(* System generated code, could be modified for your application *)
	c_udiNumberOfSubModules			: UDINT := 4;			(* Number of SubModules: Added extra 1 for Crank Module *)
	c_udiSlave3						: UDINT := 1;
	c_udiSlave4						: UDINT := 2;
	c_udiCrank						: UDINT := 4;			(* special constant for Crank module *)
	c_udiNocke1						: UDINT := 3;
(* End of system generated code, could be modified for your application *)
END_VAR

VAR (* User specific variables *)
	stSlave3Interface				: AXM.ST_ModuleInterface;
	fbSlave3Module					: AXM.FB_AxisModule;
	
	stSlave4Interface				: AXM.ST_ModuleInterface;
	fbSlave4Module					: AXM.FB_AxisModule;

	fbAxisModuleController			: AXM.FB_AxisModuleController;

	stNocke1Interface				: ST_ExampleLeafModuleInterface;
	fbNocke1Module					: FB_ExampleLeafModule;

	fbExampleLeafModuleController	: FB_ExampleLeafModuleController;
	
	(*included for CrankModule*)
	stCrankModuleItf			: CRKM.ST_ModuleInterface;
	fbCrankModule				: CRKM.FB_CrankModule;
	fbCrankModuleCtrl			: CRKM.FB_CrankModuleController;
	
	(*included for CrankModule*)
	
	xFirstCall						: BOOL := TRUE;
	iPosState						: INT := 1;
END_VAR

VAR_INPUT
(* Master of AlphaModule *)
	i_ifMaster						: SystemConfigurationItf.IF_Master;
END_VAR

VAR_IN_OUT
(* TPL.ST_StandardModuleInterface *)
	iq_stStandardModuleItf			: TPL.ST_StandardModuleInterface;
	
(* TPL.ST_StandardMotionInterface *)
	iq_stStandardMotionItf			: TPL.ST_StandardMotionInterface;
	
(* ExceptionHandling and Logging *)	
	iq_stExceptionList				: TPL.ST_ExceptionList;
	iq_stLogDataList				: TPL.ST_LogDataList;
END_VAR

VAR
	xInitSuccessful : BOOL := TRUE;
	
(* Standard related variables *)
	astSubModuleInterface			: ARRAY[1..c_udiNumberOfSubModules] OF TPL.ST_StandardModuleInterface;		(* Interface to modules *)
	aaudiSubModuleGroups			: ARRAY[1..c_udiNumberOfGroups,1..c_udiNumberOfGroupMembers] OF UDINT;
	adwSubModuleAddInterfaces		: ARRAY[1..c_udiNumberOfSubModules] OF DWORD;

(* Modules related variables *)
	fbModuleController				: TPL.FB_ModuleController;
	etDiagModuleController			: GD.ET_Diag;
	etDiagExtModuleController		: TPL.ET_DiagExt;
	sMsgModuleController			: STRING[80];
	xWaitForStartStep				: BOOL;

	astListOfCmdTables				: ARRAY [1..c_udiNumberOfCmdTables] OF TPL.ST_CmdTable;
	udiTableIndex					: UDINT;
	udiStepIndex					: UDINT;
	diStep							: DINT;

	astPrepareTable					: ARRAY [1..c_udiNumberOfCmdSteps] OF TPL.ST_Cmd;		(* Relating  Cmd table *)
	astAutoTable					: ARRAY [1..c_udiNumberOfCmdSteps] OF TPL.ST_Cmd;		(* Relating  Cmd table *)
	astManualTable					: ARRAY [1..c_udiNumberOfCmdSteps] OF TPL.ST_Cmd;		(* Relating  Cmd table *)
	astHoldTable					: ARRAY [1..c_udiNumberOfCmdSteps] OF TPL.ST_Cmd;		(* Relating  Cmd table *)
	astStartTable					: ARRAY [1..c_udiNumberOfCmdSteps] OF TPL.ST_Cmd;		(* Relating  Cmd table *)
	astStopTable					: ARRAY [1..c_udiNumberOfCmdSteps] OF TPL.ST_Cmd;		(* Relating  Cmd table *)
	astBrakeReleaseTable			: ARRAY [1..c_udiNumberOfCmdSteps] OF TPL.ST_Cmd;		(* Relating  Cmd table *)
	astAbortTable					: ARRAY [1..c_udiNumberOfCmdSteps] OF TPL.ST_Cmd;		(* Relating  Cmd table *)

(* ExceptionHandling related variables *)
	fbExceptionHandler				: TPL.FB_ExceptionHandler;

	aetReactionTranslationMode		: ARRAY[1..c_udiNumberOfSubModules] OF TPL.ET_ReactionTranslationMode;
	aastReactionTranslationTable	: ARRAY[1..c_udiNumberOfSubModules,1..TPL.Gc_udiMaxNumberOfReactions] OF TPL.ST_Reaction;
	astReactionTranslationJobs		: ARRAY[1..c_udiNumberOfSubModules] OF TPL.ST_ReactionTranslationJobs;
	
(* Exception declaration *)
	stUserException1				: TPL.ST_Exception;
	stUserException2				: TPL.ST_Exception;
	xModuleUserException1			: BOOL;
	xModuleUserException2			: BOOL;
	
	stUpdateStructsException		: TPL.ST_Exception;
	xUpdateStructsException			: BOOL;
	
	stInitReactionsException		: TPL.ST_Exception;
	xInitReactionsException			: BOOL;
	
	stInitSubModulesException		: TPL.ST_Exception;
	xInitSubModulesException		: BOOL;
	
	stIsDriveVirtualException		: TPL.ST_Exception;
	xIsDriveVirtualException		: BOOL;
	
(* Logging related variables*)
	fbLogger						: TPL.FB_Logger;

(* OnlineChange related variables *)
	fbDetectOnlineChange			: TPL.FB_DetectOnlineChange;
	xDetectOnlineChangeActive		: BOOL; 
	xDetectOnlineChangeReady		: BOOL; 
	etDetectOnlineChangeDiag		: GD.ET_Diag;
	etDetectOnlineChangeDiagExt		: TPL.ET_DiagExt; 
	sDetectOnlineChangeMsg			: STRING[80];
	
(* Init related variables *)		
	stLogicalAddressMaster			: SystemConfigurationItf.ST_LogicalAddress;
	lrShaftRefDelay					: LREAL;
	diResult						: DINT;	
	
	xDriveIsVirtual					: BOOL;	

(* POU-Feedback related variables*)	
	etDiag			: GD.ET_Diag;
	etDiagExt		: ET_DiagExt;
	etDiagDiagExtExampleLeafModule		: ET_DiagExtExampleLeafModule;
	etDiagExtTPL	: TPL.ET_DiagExt;
	etDiagExtAXM	: AXM.ET_DiagExt;
	etDiagExtCRKM	: CRKM.ET_DiagExt;
	sMsgBuffer		: STRING[80];
END_VAR

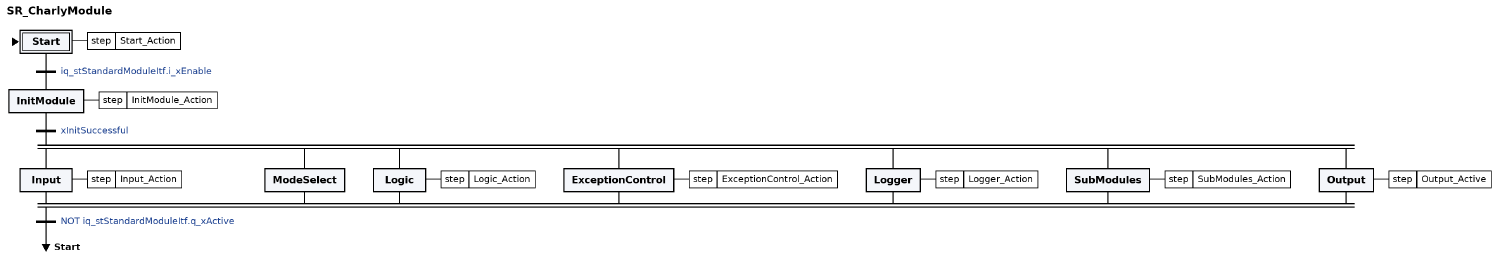
INITIAL_STEP Start:
    Start_Action(N);  // step action
END_STEP
TRANSITION FROM Start TO InitModule
    := iq_stStandardModuleItf.i_xEnable;
END_TRANSITION
STEP InitModule:
    InitModule_Action(N);  // step action
END_STEP
TRANSITION FROM InitModule TO (Input, ModeSelect, Logic, ExceptionControl, Logger, SubModules, Output)
    := xInitSuccessful;
END_TRANSITION
STEP Input:
    Input_Action(N);  // step action
END_STEP
STEP ModeSelect:
END_STEP
STEP Logic:
    Logic_Action(N);  // step action
END_STEP
STEP ExceptionControl:
    ExceptionControl_Action(N);  // step action
END_STEP
STEP Logger:
    Logger_Action(N);  // step action
END_STEP
STEP SubModules:
    SubModules_Action(N);  // step action
END_STEP
STEP Output:
    Output_Active(N);  // step action
END_STEP
TRANSITION FROM (Input, ModeSelect, Logic, ExceptionControl, Logger, SubModules, Output) TO Start
    := NOT iq_stStandardModuleItf.q_xActive;
END_TRANSITION

ACTION ExceptionControl_Action:
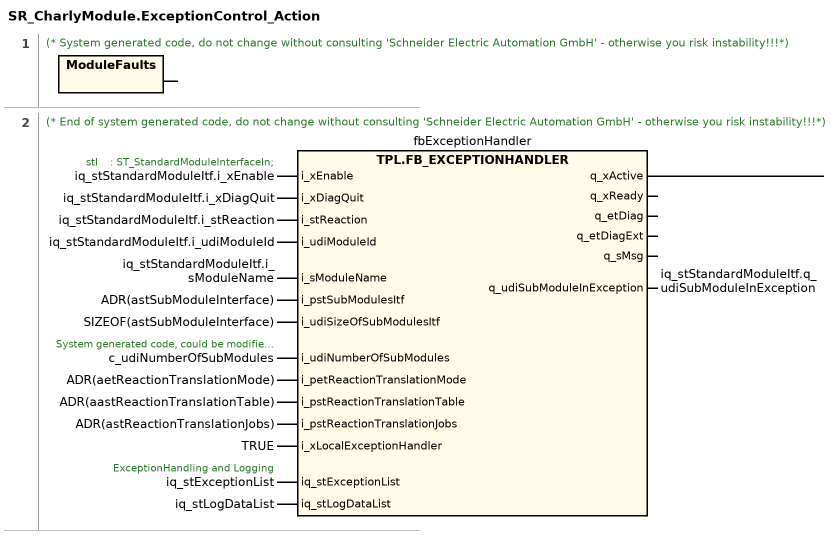
// NETWORK 1
// (* System generated code, do not change without consulting 'Schneider Electric Automation GmbH' - otherwise you risk instability!!!*)
ModuleFaults();

// NETWORK 2
// (* End of system generated code, do not change without consulting 'Schneider Electric Automation GmbH' - otherwise you risk instability!!!*)
//   fbExceptionHandler: ExceptionHandling related variables
//   iq_stStandardModuleItf.i_xEnable: stI : ST_StandardModuleInterfaceIn;
//   c_udiNumberOfSubModules: System generated code, could be modified for your application
//   iq_stExceptionList: ExceptionHandling and Logging
fbExceptionHandler(
    i_xEnable := iq_stStandardModuleItf.i_xEnable,
    i_xDiagQuit := iq_stStandardModuleItf.i_xDiagQuit,
    i_stReaction := iq_stStandardModuleItf.i_stReaction,
    i_udiModuleId := iq_stStandardModuleItf.i_udiModuleId,
    i_sModuleName := iq_stStandardModuleItf.i_sModuleName,
    i_pstSubModulesItf := ADR(astSubModuleInterface),
    i_udiSizeOfSubModulesItf := SIZEOF(astSubModuleInterface),
    i_udiNumberOfSubModules := c_udiNumberOfSubModules,
    i_petReactionTranslationMode := ADR(aetReactionTranslationMode),
    i_pstReactionTranslationTable := ADR(aastReactionTranslationTable),
    i_pstReactionTranslationJobs := ADR(astReactionTranslationJobs),
    i_xLocalExceptionHandler := TRUE,
    iq_stExceptionList := iq_stExceptionList,
    iq_stLogDataList := iq_stLogDataList,
    q_udiSubModuleInException => iq_stStandardModuleItf.q_udiSubModuleInException); // TPL.FB_EXCEPTIONHANDLER
END_ACTION

ACTION Init_CmdTables:
(* System generated code, could be modified for your application *)

(*********************************************************************************************************************)
(*** Prepare/Homing  ***)

TPL.FC_FirstStep(udiStepIndex, diStep);
astPrepareTable[udiStepIndex].sTitle					:= 'DriveEnable CrankModule';
astPrepareTable[udiStepIndex].udiModuleName				:= c_udiCrank;
astPrepareTable[udiStepIndex].diStep					:= diStep;
astPrepareTable[udiStepIndex].diCMD						:= CRKM.ET_Cmd.DriveEnableOn;
astPrepareTable[udiStepIndex].timTimeOut				:= T#0MS;
astPrepareTable[udiStepIndex].xEndCMD					:= FALSE;

TPL.FC_NextStep(udiStepIndex, diStep);
astPrepareTable[udiStepIndex].sTitle					:= 'Homing Mode CrankModule';
astPrepareTable[udiStepIndex].udiModuleName				:= c_udiCrank;
astPrepareTable[udiStepIndex].diStep					:= diStep;
astPrepareTable[udiStepIndex].diCMD						:= CRKM.ET_Cmd.Homing;
astPrepareTable[udiStepIndex].timTimeOut				:= T#0MS;
astPrepareTable[udiStepIndex].xEndCMD					:= FALSE;

TPL.FC_NextStep(udiStepIndex, diStep);
astPrepareTable[udiStepIndex].sTitle					:= 'Start CrankModule';
astPrepareTable[udiStepIndex].udiModuleName				:= c_udiCrank;
astPrepareTable[udiStepIndex].diStep					:= diStep;
astPrepareTable[udiStepIndex].diCMD						:= CRKM.ET_Cmd.Start;
astPrepareTable[udiStepIndex].timTimeOut				:= T#0MS;
astPrepareTable[udiStepIndex].xEndCMD					:= FALSE;

TPL.FC_LastStep(udiStepIndex, diStep);
astPrepareTable[udiStepIndex].sTitle					:= 'End';
astPrepareTable[udiStepIndex].udiModuleName				:= 0;
astPrepareTable[udiStepIndex].diStep					:= diStep;
astPrepareTable[udiStepIndex].diCMD						:= 0;
astPrepareTable[udiStepIndex].timTimeOut				:= T#0MS;
astPrepareTable[udiStepIndex].xEndCMD					:= TRUE;

TPL.FC_FirstCmdTable(iq_udiTableIndex:= udiTableIndex);
astListofCMDTables[udiTableIndex].sTitle				:= 'Prepare';
astListofCMDTables[udiTableIndex].diCMD					:= ET_Cmd.Prepare;
astListofCMDTables[udiTableIndex].udiNumberOfCmdSteps	:= udiStepIndex;

(*********************************************************************************************************************)
(*** Auto/Endless  ***)


TPL.FC_FirstStep(udiStepIndex, diStep);
astAutoTable[udiStepIndex].sTitle						:= 'DriveEnable CrankModule';
astAutoTable[udiStepIndex].udiModuleName				:= c_udiCrank;
astAutoTable[udiStepIndex].diStep						:= diStep;
astAutoTable[udiStepIndex].diCMD						:= CRKM.ET_Cmd.DriveEnableOn;
astAutoTable[udiStepIndex].timTimeOut					:= T#0MS;
astAutoTable[udiStepIndex].xEndCMD						:= FALSE;

TPL.FC_NextStep(udiStepIndex, diStep);
astAutoTable[udiStepIndex].sTitle						:= 'Auto/Endless CrankModule';
astAutoTable[udiStepIndex].udiModuleName				:= c_udiCrank;
astAutoTable[udiStepIndex].diStep						:= diStep;
astAutoTable[udiStepIndex].diCMD						:= CRKM.ET_Cmd.Endless;
astAutoTable[udiStepIndex].timTimeOut					:= T#0MS;
astAutoTable[udiStepIndex].xEndCMD						:= FALSE;

TPL.FC_NextStep(udiStepIndex, diStep);
astAutoTable[udiStepIndex].sTitle						:= 'Start CrankModule';
astAutoTable[udiStepIndex].udiModuleName				:= c_udiCrank;
astAutoTable[udiStepIndex].diStep						:= diStep;
astAutoTable[udiStepIndex].diCMD						:= CRKM.ET_Cmd.Start;
astAutoTable[udiStepIndex].timTimeOut					:= T#0MS;
astAutoTable[udiStepIndex].xEndCMD						:= FALSE;

TPL.FC_NextStep(udiStepIndex, diStep);
astAutoTable[udiStepIndex].sTitle						:= 'Endless Mode Slave3';
astAutoTable[udiStepIndex].udiModuleName				:= c_udiSlave3;
astAutoTable[udiStepIndex].diStep						:= diStep;
astAutoTable[udiStepIndex].diCMD						:= AXM.ET_Cmd.Endless; 
astAutoTable[udiStepIndex].timTimeOut					:= T#0MS;
astAutoTable[udiStepIndex].xEndCMD						:= FALSE;

TPL.FC_NextStep(udiStepIndex, diStep);
astAutoTable[udiStepIndex].sTitle						:= 'Positioning Mode Slave4';
astAutoTable[udiStepIndex].udiModuleName				:= c_udiSlave4;
astAutoTable[udiStepIndex].diStep						:= diStep;
astAutoTable[udiStepIndex].diCMD						:= AXM.ET_Cmd.Positioning;
astAutoTable[udiStepIndex].timTimeOut					:= T#0MS;
astAutoTable[udiStepIndex].xEndCMD						:= FALSE;

TPL.FC_NextStep(udiStepIndex, diStep);
astAutoTable[udiStepIndex].sTitle						:= 'Start Slave3';
astAutoTable[udiStepIndex].udiModuleName				:= c_udiSlave3;
astAutoTable[udiStepIndex].diStep						:= diStep;
astAutoTable[udiStepIndex].diCMD						:= AXM.ET_Cmd.Start;
astAutoTable[udiStepIndex].timTimeOut					:= T#0MS;
astAutoTable[udiStepIndex].xEndCMD						:= FALSE;



TPL.FC_LastStep(udiStepIndex, diStep);
astAutoTable[udiStepIndex].sTitle						:= 'End';
astAutoTable[udiStepIndex].udiModuleName				:= 0;
astAutoTable[udiStepIndex].diStep						:= diStep;
astAutoTable[udiStepIndex].diCMD						:= 0;
astAutoTable[udiStepIndex].timTimeOut					:= T#0MS;
astAutoTable[udiStepIndex].xEndCMD						:= TRUE;

TPL.FC_NextCmdTable(iq_udiTableIndex:= udiTableIndex);
astListofCMDTables[udiTableIndex].sTitle				:= 'Auto';
astListofCMDTables[udiTableIndex].diCMD					:= ET_Cmd.Auto;
astListofCMDTables[udiTableIndex].udiNumberOfCmdSteps	:= udiStepIndex;


(*********************************************************************************************************************)
(*** Manual  ***)

TPL.FC_FirstStep(udiStepIndex, diStep);
astManualTable[udiStepIndex].sTitle						:= 'DriveEnable On CrankModule';
astManualTable[udiStepIndex].udiModuleName				:= c_udiCrank;
astManualTable[udiStepIndex].diStep						:= diStep;
astManualTable[udiStepIndex].diCMD						:= CRKM.ET_Cmd.DriveEnableOn;
astManualTable[udiStepIndex].timTimeOut					:= T#0MS;
astManualTable[udiStepIndex].xEndCMD					:= FALSE;

TPL.FC_NextStep(udiStepIndex, diStep);
astManualTable[udiStepIndex].sTitle						:= 'Manual Mode CrankModule';
astManualTable[udiStepIndex].udiModuleName				:= c_udiCrank;
astManualTable[udiStepIndex].diStep						:= diStep;
astManualTable[udiStepIndex].diCMD						:= CRKM.ET_Cmd.Manual;
astManualTable[udiStepIndex].timTimeOut					:= T#0MS;
astManualTable[udiStepIndex].xEndCMD					:= FALSE;

TPL.FC_LastStep(udiStepIndex, diStep);
astManualTable[udiStepIndex].sTitle						:= 'End';
astManualTable[udiStepIndex].udiModuleName				:= 0;
astManualTable[udiStepIndex].diStep						:= diStep;
astManualTable[udiStepIndex].diCMD						:= 0;
astManualTable[udiStepIndex].timTimeOut					:= T#0MS;
astManualTable[udiStepIndex].xEndCMD					:= TRUE;

TPL.FC_NextCmdTable(iq_udiTableIndex:= udiTableIndex);
astListofCMDTables[udiTableIndex].sTitle				:= 'Manual';
astListofCMDTables[udiTableIndex].diCMD					:= ET_Cmd.Manual;
astListofCMDTables[udiTableIndex].udiNumberOfCmdSteps	:= udiStepIndex;

(*********************************************************************************************************************)
(*** Stop ***)

TPL.FC_FirstStep(udiStepIndex, diStep);
astStopTable[udiStepIndex].sTitle						:= 'Stop CrankModule';
astStopTable[udiStepIndex].udiModuleName				:= c_udiCrank;
astStopTable[udiStepIndex].diStep						:= diStep;
astStopTable[udiStepIndex].diCMD						:= CRKM.ET_Cmd.Stop;
astStopTable[udiStepIndex].timTimeOut					:= T#0MS;
astStopTable[udiStepIndex].xEndCMD						:= FALSE;

TPL.FC_LastStep(udiStepIndex, diStep);
astStopTable[udiStepIndex].sTitle						:= 'End';
astStopTable[udiStepIndex].udiModuleName				:= 0;
astStopTable[udiStepIndex].diStep						:= diStep;
astStopTable[udiStepIndex].diCMD						:= 0;
astStopTable[udiStepIndex].timTimeOut					:= T#0MS;
astStopTable[udiStepIndex].xEndCMD						:= TRUE;

TPL.FC_NextCmdTable(iq_udiTableIndex:= udiTableIndex);
astListofCMDTables[udiTableIndex].sTitle				:= 'Stop';
astListofCMDTables[udiTableIndex].diCMD					:= ET_Cmd.Stop;
astListofCMDTables[udiTableIndex].udiNumberOfCmdSteps	:= udiStepIndex;

(*********************************************************************************************************************)
(*** Start ***)

TPL.FC_FirstStep(udiStepIndex, diStep);
astStartTable[udiStepIndex].sTitle						:= 'Start CrankModule';
astStartTable[udiStepIndex].udiModuleName				:= c_udiCrank;
astStartTable[udiStepIndex].diStep						:= diStep;
astStartTable[udiStepIndex].diCMD						:= CRKM.ET_Cmd.Start;
astStartTable[udiStepIndex].timTimeOut					:= T#0MS;
astStartTable[udiStepIndex].xEndCMD						:= FALSE;

TPL.FC_LastStep(udiStepIndex, diStep);
astStartTable[udiStepIndex].sTitle						:= 'End';
astStartTable[udiStepIndex].udiModuleName				:= 0;
astStartTable[udiStepIndex].diStep						:= diStep;
astStartTable[udiStepIndex].diCMD						:= 0;
astStartTable[udiStepIndex].timTimeOut					:= T#0MS;
astStartTable[udiStepIndex].xEndCMD						:= TRUE;

TPL.FC_NextCmdTable(iq_udiTableIndex:= udiTableIndex);
astListofCMDTables[udiTableIndex].sTitle				:= 'Start';
astListofCMDTables[udiTableIndex].diCMD					:= ET_Cmd.Start;
astListofCMDTables[udiTableIndex].udiNumberOfCmdSteps	:= udiStepIndex;

(*********************************************************************************************************************)
(*** Abort ***)

TPL.FC_FirstStep(udiStepIndex, diStep);
astAbortTable[udiStepIndex].sTitle						:= 'Stop CrankModule';
astAbortTable[udiStepIndex].udiModuleName				:= c_udiCrank;
astAbortTable[udiStepIndex].diStep						:= diStep;
astAbortTable[udiStepIndex].diCMD						:= CRKM.ET_Cmd.Stop;
astAbortTable[udiStepIndex].timTimeOut					:= T#0MS;
astAbortTable[udiStepIndex].xEndCMD						:= FALSE;

TPL.FC_LastStep(udiStepIndex, diStep);
astAbortTable[udiStepIndex].sTitle						:= 'End';
astAbortTable[udiStepIndex].udiModuleName				:= 0;
astAbortTable[udiStepIndex].diStep						:= diStep;
astAbortTable[udiStepIndex].diCMD						:= 0;
astAbortTable[udiStepIndex].timTimeOut					:= T#0MS;
astAbortTable[udiStepIndex].xEndCMD						:= TRUE;

TPL.FC_NextCmdTable(iq_udiTableIndex:= udiTableIndex);
astListofCMDTables[udiTableIndex].sTitle				:= 'Abort';
astListofCMDTables[udiTableIndex].diCMD					:= ET_Cmd.Abort;
astListofCMDTables[udiTableIndex].udiNumberOfCmdSteps	:= udiStepIndex;

(*********************************************************************************************************************)
(*** Hold ***)

TPL.FC_FirstStep(udiStepIndex, diStep);
astHoldTable[udiStepIndex].sTitle						:= 'Hold CrankModule';
astHoldTable[udiStepIndex].udiModuleName				:= c_udiCrank;
astHoldTable[udiStepIndex].diStep						:= diStep;
astHoldTable[udiStepIndex].diCMD						:= CRKM.ET_Cmd.Hold;
astHoldTable[udiStepIndex].timTimeOut					:= T#0MS;
astHoldTable[udiStepIndex].xEndCMD						:= FALSE;

TPL.FC_NextStep(udiStepIndex, diStep);
astHoldTable[udiStepIndex].sTitle						:= 'Hold_Slave3';
astHoldTable[udiStepIndex].udiModuleName				:= c_udiSlave3;
astHoldTable[udiStepIndex].diStep						:= diStep;
astHoldTable[udiStepIndex].diCMD						:= AXM.ET_Cmd.Hold;
astHoldTable[udiStepIndex].timTimeOut					:= T#0MS;
astHoldTable[udiStepIndex].xEndCMD						:= FALSE;

TPL.FC_NextStep(udiStepIndex, diStep);
astHoldTable[udiStepIndex].sTitle						:= 'Stop_Slave4';
astHoldTable[udiStepIndex].udiModuleName				:= c_udiSlave4;
astHoldTable[udiStepIndex].diStep						:= diStep;
astHoldTable[udiStepIndex].diCMD						:= AXM.ET_Cmd.Stop;
astHoldTable[udiStepIndex].timTimeOut					:= T#0MS;
astHoldTable[udiStepIndex].xEndCMD						:= FALSE;

TPL.FC_LastStep(udiStepIndex, diStep);
astHoldTable[udiStepIndex].sTitle						:= 'End';
astHoldTable[udiStepIndex].udiModuleName				:= 0;
astHoldTable[udiStepIndex].diStep						:= diStep;
astHoldTable[udiStepIndex].diCMD						:= 0;
astHoldTable[udiStepIndex].timTimeOut					:= T#0MS;
astHoldTable[udiStepIndex].xEndCMD						:= TRUE;

TPL.FC_NextCmdTable(iq_udiTableIndex:= udiTableIndex);
astListofCMDTables[udiTableIndex].sTitle				:= 'Hold';
astListofCMDTables[udiTableIndex].diCMD					:= ET_Cmd.Hold;
astListofCMDTables[udiTableIndex].udiNumberOfCmdSteps	:= udiStepIndex;

(*********************************************************************************************************************)
(*** Brake Release ***)

TPL.FC_FirstStep(udiStepIndex, diStep);
astBrakeReleaseTable[udiStepIndex].sTitle				:= 'DriveEnable Off CrankModule';
astBrakeReleaseTable[udiStepIndex].udiModuleName		:= c_udiCrank;
astBrakeReleaseTable[udiStepIndex].diStep				:= diStep;
astBrakeReleaseTable[udiStepIndex].diCMD				:= CRKM.ET_Cmd.DriveEnableOff;
astBrakeReleaseTable[udiStepIndex].timTimeOut			:= T#0MS;
astBrakeReleaseTable[udiStepIndex].xEndCMD				:= FALSE;

TPL.FC_NextStep(udiStepIndex, diStep);
astBrakeReleaseTable[udiStepIndex].sTitle				:= 'BrakeRelease Mode CrankModule';
astBrakeReleaseTable[udiStepIndex].udiModuleName		:= c_udiCrank;
astBrakeReleaseTable[udiStepIndex].diStep				:= diStep;
astBrakeReleaseTable[udiStepIndex].diCMD				:= CRKM.ET_Cmd.BrakeRelease;
astBrakeReleaseTable[udiStepIndex].timTimeOut			:= T#0MS;
astBrakeReleaseTable[udiStepIndex].xEndCMD				:= FALSE;

TPL.FC_NextStep(udiStepIndex, diStep);
astBrakeReleaseTable[udiStepIndex].sTitle				:= 'Start CrankModule';
astBrakeReleaseTable[udiStepIndex].udiModuleName		:= c_udiCrank;
astBrakeReleaseTable[udiStepIndex].diStep				:= diStep;
astBrakeReleaseTable[udiStepIndex].diCMD				:= CRKM.ET_Cmd.Start;
astBrakeReleaseTable[udiStepIndex].timTimeOut			:= T#0MS;
astBrakeReleaseTable[udiStepIndex].xEndCMD				:= FALSE;

TPL.FC_LastStep(udiStepIndex, diStep);
astBrakeReleaseTable[udiStepIndex].sTitle				:= 'End';
astBrakeReleaseTable[udiStepIndex].udiModuleName		:= 0;
astBrakeReleaseTable[udiStepIndex].diStep				:= diStep;
astBrakeReleaseTable[udiStepIndex].diCMD				:= 0;
astBrakeReleaseTable[udiStepIndex].timTimeOut			:= T#0MS;
astBrakeReleaseTable[udiStepIndex].xEndCMD				:= TRUE;

TPL.FC_NextCmdTable(iq_udiTableIndex:= udiTableIndex);
astListofCMDTables[udiTableIndex].sTitle				:= 'Brake Release';
astListofCMDTables[udiTableIndex].diCMD					:= ET_Cmd.BrakeRelease;
astListofCMDTables[udiTableIndex].udiNumberOfCmdSteps	:= udiStepIndex;

(* End of system generated code, could be modified for your application *)
END_ACTION

ACTION Init_CrankModule:
(* Standard interface *)
astSubModuleInterface[c_udiCrank].i_sModuleName:= Standard.CONCAT(STR1:= iq_stStandardModuleItf.i_sModuleName, STR2:= ': CrankModule');

(*
	Crank module interface 
*)

stCrankModuleItf.stMain.i_ifDriveCrank			:= DRV_CrankDrive;
stCrankModuleItf.stMain.iq_lencEncoderCrank		:= LE_EncCrank;

stCrankModuleItf.stMain.i_ifDriveSlide			:= DRV_SlideDrive;
stCrankModuleItf.stMain.iq_lencEncoderSlide		:= LE_EncSlide;

stCrankModuleItf.stMain.i_ifMaster				:= DRV_Master;


stCrankModuleItf.stMain.i_lrMotionActiveVelLimit	:= 15.0;		(* Limit for max. velocity of astAxisModuleInterface  to switch output AxisMove in Units/s *)
stCrankModuleItf.stMain.i_etMotionActiveVelType		:= CRKM.ET_MotionActiveVelType.RefVelocity;


(***************************************************************************************************************************************************************************************************)
(*** Homing ***)

stCrankModuleItf.stHome.stTouchProbe.i_ifTouchProbe	:= TP_1;

stCrankModuleItf.stHome.i_etMode					:= PDL.ET_HomeMode.SetPosAxisAndLogEncoderPosition;	(* Homing Mode in case of real axis *)

stCrankModuleItf.stHome.i_xEnableInitAbsReadPos		:= FALSE;
																			(* TRUE : Restores the AxisPosition depending on the stHome.etMode
																			 if stHome.etMode is equal PDL.ET_HomeMode.RestorePosFromAxisencoder or 
																			 PDL.ET_HomeMode.WriteAxisEncoder, the encoder of the axis is read,
																			 or else the position will be restored from the retain area*)
stCrankModuleItf.stHome.stSetpos.iq_pstRestorePosRetain	:= ADR(Grp_stRestorePositionAxisCrank);

(* Possible modes for homing mode Sensor:
	PDL.ET_HomeMode.PosDirectionPosEdgeSensor
	PDL.ET_HomeMode.NegDirectionPosEdgeSensor
	PDL.ET_HomeMode.NegDirectionNegEdgeSensor
	PDL.ET_HomeMode.PosDirectionNegEdgeSensor
*)
stCrankModuleItf.stHome.stSensor.i_lrHomePosition		:= 0.0;			(* Position at the end of homing in units *)
stCrankModuleItf.stHome.stSensor.i_lrVel				:= 10.0;		(* Homing ceiling velocity in units/s *)
stCrankModuleItf.stHome.stSensor.i_lrAcc				:= 1000.0;		(* Homing acceleration in units/s^2 *)
stCrankModuleItf.stHome.stSensor.i_lrDec				:= 1000.0;		(* Homing deceleration in units/s^2 *)
stCrankModuleItf.stHome.stSensor.i_lrJerk				:= 100000.0;	(* Homing jerk in units/s^3 *)
stCrankModuleItf.stHome.stSensor.i_lrOffset				:= 0.0;			(* Offset from home signal in units *)
stCrankModuleItf.stHome.stSensor.i_lrMaxTravel			:= 720.0;		(* Max. travel for refering by  normal input *)
stCrankModuleItf.stHome.stSensor.i_xRotativeSystem		:= FALSE;		(* Rotative system true or false for refering by normal input *)

(* Possible Modes for homing mode LimitSwitch:
	PDL.ET_HomeMode.PosDirectionPosEdgeHWLimitPos		normally open contact / Closing contact
	PDL.ET_HomeMode.NegDirectionPosEdgeHWLimitNeg		normally open contact / Closing contact
	PDL.ET_HomeMode.NegDirectionNegEdgeHWLimitNeg		normally closed contact / Opening contact  
	PDL.ET_HomeMode.PosDirectionNegEdgeHWLimitPos		normally closed contact / Opening contact 
*)
stCrankModuleItf.stHome.stLimitSwitch.i_lrHomePosition	:= 0.0;			(* Position at the end of homing in units *)
stCrankModuleItf.stHome.stLimitSwitch.i_lrVel			:= 10.0;		(* Homing ceiling velocity in units/s *)
stCrankModuleItf.stHome.stLimitSwitch.i_lrAcc			:= 1000.0;		(* Homing acceleration in units/s^2 *)
stCrankModuleItf.stHome.stLimitSwitch.i_lrDec			:= 1000.0;		(* Homing deceleration in units/s^2 *)
stCrankModuleItf.stHome.stLimitSwitch.i_lrOffset		:= 0.0;			(* Offset from home signal in units *)
stCrankModuleItf.stHome.stLimitSwitch.i_lrMaxTravel		:= 9999.0;		(* Max. travel for referencing normal input as a hardware limit *)
stCrankModuleItf.stHome.stLimitSwitch.i_lrJerk			:= 1000000.0;	(* Homing jerk in units/s^3 *)

(* Possible modes for homing mode MoveOnPos:
	PDL.ET_HomeMode.MoveOnPosAbs 
*)
stCrankModuleItf.stHome.stMoveonPos.i_lrTarget			:= 0.0;			(* Position at the end of homing in units *)
stCrankModuleItf.stHome.stMoveonPos.i_lrVel				:= 10.0;		(* Homing ceiling velocity in units/s *)
stCrankModuleItf.stHome.stMoveonPos.i_lrAcc				:= 1000.0;		(* Homing acceleration in units/s^2 *)
stCrankModuleItf.stHome.stMoveonPos.i_lrDec				:= 1000.0;		(* Homing deceleration in units/s^2 *)
stCrankModuleItf.stHome.stMoveonPos.i_xRotativeSystem	:= FALSE;		(* Rotative system true or false *)
stCrankModuleItf.stHome.stMoveonPos.i_lrPeriod			:= 0.0;			(* Period of the axis *)
stCrankModuleItf.stHome.stMoveonPos.i_lrJerk			:= 1000000.0;	(* Homing jerk in units/s^3 *)

(* Possible modes for homing mode SetPos:
	PDL.ET_HomeMode.SetPosAxisPosition 
	PDL.ET_HomeMode.SetPosLogEncoderPosition 
	PDL.ET_HomeMode.SetPosAxisAndLogEncoderPosition
	PDL.ET_HomeMode.RestorePosFromAxisEncoder 
	PDL.ET_HomeMode.RestorePosFromRetain 
*)
stCrankModuleItf.stHome.stSetpos.i_lrHomePosition		:= 100.0;		(* Position at the end of homing in units *)
stCrankModuleItf.stHome.stSetpos.i_lrEncoderPosition	:= 0.0;			(* Encoder position in units after homing *)
stCrankModuleItf.stHome.stSetpos.i_lrAbsEncOffset		:= 100.0;		(* Distance to the jump of axis encoder in units  *)
stCrankModuleItf.stHome.stSetpos.i_lrRestoreWindow		:= 180;			(* How far can the drive be away from is correct position *)
stCrankModuleItf.stHome.stSetpos.i_lrUserPeriod			:= 360;			(* Period of the axis *)

(* Possible modes for homing mode Torque:
	PDL.ET_HomeMode.PosDirectionMaxTorque 
	PDL.ET_HomeMode.NegDirectionMaxTorque 
*)
stCrankModuleItf.stHome.stTorque.i_lrHomePosition		:= 0.0;			(* Position at the end of homing in units *)
stCrankModuleItf.stHome.stTorque.i_lrVel				:= 10.0;		(* Homing ceiling velocity in units/s *)
stCrankModuleItf.stHome.stTorque.i_lrAcc				:= 1000.0;		(* Homing acceleration in units/s^2 *)
stCrankModuleItf.stHome.stTorque.i_lrDec				:= 1000.0;		(* Homing deceleration in units/s^2 *)
stCrankModuleItf.stHome.stTorque.i_lrOffset				:= 0.0;			(* Offset from home signal in units *)
stCrankModuleItf.stHome.stTorque.i_lrMaxTravel			:= 9999.0;		(* Max. travel for referencing by TP or normal input *)
stCrankModuleItf.stHome.stTorque.i_lrMaxTorque			:= 0.0;			(* Torque for stop in Nm / referencing by torque *)
stCrankModuleItf.stHome.stTorque.i_lrJerk				:= 1000000.0;	(* Homing jerk in units/s^3 *)
stCrankModuleItf.stHome.stTorque.i_diTorqueTime			:= 5;			(* Time in msec to hold torque *)

(* Possible modes for homing mode TouchProbe:
	PDL.ET_HomeMode.PosDirectionPosEdgeTp 
	PDL.ET_HomeMode.NegDirectionPosEdgeTp 
	PDL.ET_HomeMode.NegDirectionNegEdgeTp 
	PDL.ET_HomeMode.PosDirectionNegEdgeTp 
*)
stCrankModuleItf.stHome.stTouchProbe.i_lrHomePosition	:= 0.0;			(* Position at the end of homing in units *)
stCrankModuleItf.stHome.stTouchProbe.i_lrVel			:= 100.0;		(* Homing ceiling velocity in units/s *)
stCrankModuleItf.stHome.stTouchProbe.i_lrAcc			:= 1000.0;		(* Homing acceleration in units/s^2 *)
stCrankModuleItf.stHome.stTouchProbe.i_lrDec			:= 1000.0;		(* Homing deceleration in units/s^2 *)
stCrankModuleItf.stHome.stTouchProbe.i_lrOffset			:= 30.0;		(* Offset from home signal in units *)
stCrankModuleItf.stHome.stTouchProbe.i_lrMaxTravel		:= 720.0;		(* Max. travel for referencing by TP or normal input *)
stCrankModuleItf.stHome.stTouchProbe.i_xRotativeSystem	:= TRUE;		(* Rotative system true or false for referencing by TP *)
stCrankModuleItf.stHome.stTouchProbe.i_lrJerk			:= 1000000.0;	(* Homing jerk in units/s^3 *)

(* Possible modes for HomeWritePos:
	PDL.ET_HomeMode.WriteAxisEncoder
*)
stCrankModuleItf.stHome.stWritePos.i_lrHomePosition		:= 0.0;			(* Position at the end of homing in units *)
stCrankModuleItf.stHome.stWritePos.i_lrUserPeriod		:= 0.0;			(* Calculates Drive.position into period ( units ) *)
stCrankModuleItf.stHome.stWritePos.i_lrAbsEncOffset		:= 180.0;		(* Distance to the jump of axis encoder in units *)

(***************************************************************************************************************************************************************************************************)
(*** Manual ***)
stCrankModuleItf.stManual.i_xCrankMode					:= FALSE;			(* TRUE: Jogging CrankAxis, FALSE: Jogging SlideAxis *)
stCrankModuleItf.stManual.i_lrVel						:= 25.0;			(* Velocity in units/s *)
stCrankModuleItf.stManual.i_lrAcc						:= 100.0;			(* Acceleration in units/s^2 *)
stCrankModuleItf.stManual.i_lrDec						:= 100.0;			(* Deceleration in units/s^2 *)
stCrankModuleItf.stManual.i_lrMaxDistance				:= 120.0;			(* Max pathlengths for one step in units *)
stCrankModuleItf.stManual.i_xEndless					:= FALSE;			(* TRUE: jogging endless; Position between the periode; FALSE: jogging in steps. Position can be out of periode *)
stCrankModuleItf.stManual.i_lrJerk						:= 10000.0;			(* Jerk in units/s^3 *)

(***************************************************************************************************************************************************************************************************)
(*** Cam ***)

stCrankModuleItf.stMultiCam.i_etCSModeSlave				:= PDL.ET_MultiCamCsModeSlave.SetSlavePositionToFirstCamPosition;	(* ColdStartMode Axis *)
stCrankModuleItf.stMultiCam.i_etCSModeMaster			:= PDL.ET_MultiCamCsModeMaster.SetMasterPositionToFirstCamPosition;	(* ColdStartMode Master *)
stCrankModuleItf.stMultiCam.i_etWSMode					:= PDL.ET_MultiCamWsMode.StoredCamMoveAlwaysNoPositionCheck;		(* WarmStartMode *)
stCrankModuleItf.stMultiCam.i_lrWSWindow				:= 5.0;								(* WarmStartWindow in Axis units *)
stCrankModuleItf.stMultiCam.i_lrWSVel					:= 100.0;							(* Velocity for WarmStart and CSModeAxis = 2 in Units/s *)
stCrankModuleItf.stMultiCam.i_lrWSAcc					:= 1000.0;							(* Acceleration and deceleration for Warmstart  and CSModeAxis = 2 in Units/s2 *)
stCrankModuleItf.stMultiCam.i_lrWSJerk					:= 10000.0;
stCrankModuleItf.stMultiCam.i_diTXend					:= 2 * SystemInterface.FC_LzsTaskGetInterval();			(* Time of XLowEnd and XHighEnd befor Xend or Xstart in msec*)
stCrankModuleItf.stMultiCam.i_lrInstantXLimMax			:= 0.0;								(* Switch off position at 'InstantNewCam' *)

stCrankModuleItf.stMultiCam.i_xEnableTabHandler			:= TRUE;
stCrankModuleItf.stMultiCam.i_udiTableSelectNr			:= DINT_TO_UDINT(CRKM.ET_ParId.User);

stCrankModuleItf.stMultiCam.i_xSetEncoderParameters		:= FALSE;										(* TRUE: The parameters MasterId, FeedConstand, GearIn and GearOut will be copyed into LEnc object *)
stCrankModuleItf.stMultiCam.i_xSetEncoderPosition		:= FALSE;										(* TRUE: Manipulation of LEnc object on startup OpMode MultiCam *)
stCrankModuleItf.stMultiCam.i_lrSetEncoderOffset		:= 0.0;											(* Master encoder offset *)
stCrankModuleItf.stMultiCam.i_xCheckEncoderPeriod		:= TRUE;										(* TRUE: Check of encoder period = 0. If encoder period <> 0 -> Exception *)

stCrankModuleItf.stMultiCam.iq_astMotionPar[CRKM.ET_ParId.User].diNumberOfCamPoints			:= 4;	(* DataStruct for the next cycle *)
stCrankModuleItf.stMultiCam.iq_astMotionPar[CRKM.ET_ParId.User].lrYPeriod					:= 0.0;

stCrankModuleItf.stMultiCam.iq_astMotionPar[CRKM.ET_ParId.User].astCamPoint[0].lrX			:= 0.0;
stCrankModuleItf.stMultiCam.iq_astMotionPar[CRKM.ET_ParId.User].astCamPoint[0].lrY			:= 0.0;
stCrankModuleItf.stMultiCam.iq_astMotionPar[CRKM.ET_ParId.User].astCamPoint[0].lrM			:= 0.0;
stCrankModuleItf.stMultiCam.iq_astMotionPar[CRKM.ET_ParId.User].astCamPoint[0].etCamType	:= PDL.ET_CamType.Poly5Com;
stCrankModuleItf.stMultiCam.iq_astMotionPar[CRKM.ET_ParId.User].astCamPoint[1].lrX			:= 60.0;
stCrankModuleItf.stMultiCam.iq_astMotionPar[CRKM.ET_ParId.User].astCamPoint[1].lrY			:= 30.0;
stCrankModuleItf.stMultiCam.iq_astMotionPar[CRKM.ET_ParId.User].astCamPoint[1].lrM			:= 1.0;
stCrankModuleItf.stMultiCam.iq_astMotionPar[CRKM.ET_ParId.User].astCamPoint[1].etCamType	:= PDL.ET_CamType.Straight;
stCrankModuleItf.stMultiCam.iq_astMotionPar[CRKM.ET_ParId.User].astCamPoint[2].lrX			:= 240.0;
stCrankModuleItf.stMultiCam.iq_astMotionPar[CRKM.ET_ParId.User].astCamPoint[2].lrY			:= 210.0;
stCrankModuleItf.stMultiCam.iq_astMotionPar[CRKM.ET_ParId.User].astCamPoint[2].lrM			:= 1.0;
stCrankModuleItf.stMultiCam.iq_astMotionPar[CRKM.ET_ParId.User].astCamPoint[2].etCamType	:= PDL.ET_CamType.Poly5Com;
stCrankModuleItf.stMultiCam.iq_astMotionPar[CRKM.ET_ParId.User].astCamPoint[3].lrX			:= 360.0;
stCrankModuleItf.stMultiCam.iq_astMotionPar[CRKM.ET_ParId.User].astCamPoint[3].lrY			:= 0.0;
stCrankModuleItf.stMultiCam.iq_astMotionPar[CRKM.ET_ParId.User].astCamPoint[3].lrM			:= 0.0;
stCrankModuleItf.stMultiCam.iq_astMotionPar[CRKM.ET_ParId.User].astCamPoint[3].etCamType	:= PDL.ET_CamType.Poly5Com;

stCrankModuleItf.stMultiCam.iq_astMotionPar[CRKM.ET_ParId.Idle].diUserTableId				:= CRKM.ET_ParId.Idle;
stCrankModuleItf.stMultiCam.iq_astMotionPar[CRKM.ET_ParId.Start].diUserTableId				:= CRKM.ET_ParId.Start;
stCrankModuleItf.stMultiCam.iq_astMotionPar[CRKM.ET_ParId.Cont].diUserTableId				:= CRKM.ET_ParId.Cont;
stCrankModuleItf.stMultiCam.iq_astMotionPar[CRKM.ET_ParId.Stop].diUserTableId				:= CRKM.ET_ParId.Stop;
stCrankModuleItf.stMultiCam.iq_astMotionPar[CRKM.ET_ParId.User].diUserTableId				:= CRKM.ET_ParId.User;

(***************************************************************************************************************************************************************************************************)
(*** Endless ***)

(* ENDLESS parameters need to remain at sensible values so that it reaches a velocity of at least 10.0 within 100ms*)
stCrankModuleItf.stEndless.i_lrVel				:= 100.0;			(* Velocity in units/s *)
stCrankModuleItf.stEndless.i_lrAcc				:= 1000.0;			(* Acceleration in units/s^2 *)
stCrankModuleItf.stEndless.i_lrDec				:= 1000.0;			(* Deceleration in units/s^2 *)
stCrankModuleItf.stEndless.i_lrPeriod			:= 360.0;			(* Period one cycle in units *)
stCrankModuleItf.stEndless.i_lrStopPosition		:= 0.5;				(* Stop position in units ( if G_eStart = FALSE ) *)
stCrankModuleItf.stEndless.i_lrJerk				:= 10000.0;

(***************************************************************************************************************************************************************************************************)
(*** Pos ***)

stCrankModuleItf.stPos.i_etPosMode				:= SystemInterface.ET_PosMode.Relative;			(* POS_ENDLESS, POS_RELATIVE, POS_ABSOLUTE *)
stCrankModuleItf.stPos.i_lrTarget				:= -360.0;					(* Target position or distance in units *)
stCrankModuleItf.stPos.i_lrVel					:= 100.0;					(* Ceiling velocity in units/s *)
stCrankModuleItf.stPos.i_lrAcc					:= 3600.0;					(* Acceleration in units/s^2 *)
stCrankModuleItf.stPos.i_lrDec					:= 3600.0;					(* Deceleration in units/s^2 *)
stCrankModuleItf.stPos.i_lrJerk					:= 99999.0;					(* Jerk in units/s^3 *)

(***************************************************************************************************************************************************************************************************)
(*** Crank Transformation Data 																																									 ***)
(***************************************************************************************************************************************************************************************************)

stCrankModuleItf.stCrank.lrRadius											:= 50.0;	(* Crank radius *)
stCrankModuleItf.stCrank.lrPushRod											:= 157.2;	(* Length *)
stCrankModuleItf.stCrank.lrOffset											:= 0.0;	(* Distance crank center to slide level *)
stCrankModuleItf.stCrank.lrXStart											:= 7.2;	(* Distance crank center to 0-position of slide *)
																			
stCrankModuleItf.stCrank.diXLogEqualXMechRange	:= 1;			(* Range where logical position equals mechanical position of slide *)

stCrankModuleItf.stCrank.xCrankLeft											:= FALSE;	(* TRUE = Crank on the left hand side *)
																						(* FALSE = Crank on the right hand side *)

stCrankModuleItf.stCrank.xRange												:= FALSE;	(* if TRUE and two ranges, then take range 1 *)
																						(* if FALSE and two ranges, then take range 2 *)

stCrankModuleItf.stCrank.lrP5Pole1IntervalLow	:= 0.5;	(* Distance X pole 1 <-> low end of interpolation interval *)
stCrankModuleItf.stCrank.lrP5Pole1IntervalHigh	:= 0.5;	(* Distance X pole 1 <-> high end of interpolation interval *)
stCrankModuleItf.stCrank.lrP5Pole2IntervalLow	:= 0.5;	(* Distance X pole 2 <-> low end of interpolation interval *)
stCrankModuleItf.stCrank.lrP5Pole2IntervalHigh	:= 0.5;	(* Distance X pole 2 <-> high end of interpolation interval *)
stCrankModuleItf.stCrank.lrP5RangeLow			:= 2.0;	(* only for overlapping interpolation intervals: definition range of start polynomial *)
stCrankModuleItf.stCrank.lrP5RangeHigh			:= 2.0;	(* only for overlapping interpolation intervals: definition range of end polynomial *)

stCrankModuleItf.stCrank.lrUserMechPosOffset	:= 0.0;		(* Offset for user-defined mechanical crank position *)
stCrankModuleItf.stCrank.lrUserMechPosDirection	:= 1.0;		(* Direction for user-defined mechanical crank position *)

(* Calculated mechanical crank data *)
stCrankModuleItf.stCrank.diNumberOfRanges		:= 0;			(* in certain mechanical configurations it is possible to have two ranges *)
stCrankModuleItf.stCrank.xEndlessCrank			:= FALSE;		(* TRUE, if the mechanical configuration of the crank permits a full turn, FALSE otherwise *)
stCrankModuleItf.stCrank.lrXMechMin				:= 0;			(* Low end of linearized forward move *)
stCrankModuleItf.stCrank.lrXMechMax				:= 0;			(* High end of linearized forward move *)
stCrankModuleItf.stCrank.lrPhiMin				:= 0;			(* Crank angle for Xmin *)
stCrankModuleItf.stCrank.lrPhiMax				:= 0;			(* Crank angle for Xmax *)
stCrankModuleItf.stCrank.lrPhiXMechMin			:= 0;			(* Crank angle for XMechMin *)
stCrankModuleItf.stCrank.lrPhiXMechMax			:= 0;			(* Crank angle for XMechMax  *)

(* Calculated logical crank data *)
stCrankModuleItf.stCrank.lrXLogMin				:= 0;
stCrankModuleItf.stCrank.lrXLogSwitch			:= 0;
stCrankModuleItf.stCrank.lrXLogMax				:= 0;
stCrankModuleItf.stCrank.lrPhiLogMin			:= 0;
stCrankModuleItf.stCrank.lrPhiLogSwitch			:= 0;
stCrankModuleItf.stCrank.lrPhiLogMax			:= 0;
stCrankModuleItf.stCrank.xXLogDirPos			:= FALSE;

(* Calculated P5 data *)
stCrankModuleItf.stCrank.diP5NumberOfPoles		:= 0;

(* Internal Data *)
stCrankModuleItf.stCrank.xValidData				:= FALSE;		(* Set if calculation was ok *)
stCrankModuleItf.stCrank.xSynchron				:= FALSE;

(* End of system generated code, could be modified for your application*)
END_ACTION

ACTION Init_Exceptions:
(* System generated code, could be modified for your application *)
stUpdateStructsException.etDiag												:= GD.ET_Diag.UnexpectedProgramBehavior;
stUpdateStructsException.udiDiagExt											:= ET_DiagExt.UpdateStructsException;
stUpdateStructsException.sDiagExt											:= FC_EtDiagExtToString(i_etDiagExt := stUpdateStructsException.udiDiagExt);
stUpdateStructsException.sMsg												:= '';	(* Replaced on usage *)
stUpdateStructsException.udiModuleId										:= iq_stStandardModuleItf.i_udiModuleId;
stUpdateStructsException.sModuleName										:= iq_stStandardModuleItf.i_sModuleName;
stUpdateStructsException.stReaction.axReaction[TPL.ET_Reaction.AsyncStop]	:= TRUE;
stUpdateStructsException.etSource											:= TPL.ET_ExceptionSource.NodeModule;
stUpdateStructsException.timDelayTime										:= T#0MS;
stUpdateStructsException.wHmiAttributes										:= 0;
stUpdateStructsException.xAutoQuit											:= FALSE;

stInitReactionsException.etDiag												:= GD.ET_Diag.UnexpectedProgramBehavior;
stInitReactionsException.udiDiagExt											:= ET_DiagExt.InitReactionsException;
stInitReactionsException.sDiagExt											:= FC_EtDiagExtToString(i_etDiagExt := stInitReactionsException.udiDiagExt);
stInitReactionsException.sMsg												:= '';	(* Replaced on usage *)
stInitReactionsException.udiModuleId										:= iq_stStandardModuleItf.i_udiModuleId;
stInitReactionsException.sModuleName										:= iq_stStandardModuleItf.i_sModuleName;
stInitReactionsException.stReaction.axReaction[TPL.ET_Reaction.AsyncStop]	:= TRUE;
stInitReactionsException.etSource											:= TPL.ET_ExceptionSource.NodeModule;
stInitReactionsException.timDelayTime										:= T#0MS;
stInitReactionsException.wHmiAttributes										:= 0;
stInitReactionsException.xAutoQuit											:= FALSE;

stInitSubModulesException.etDiag											:= GD.ET_Diag.UnexpectedProgramBehavior;
stInitSubModulesException.udiDiagExt										:= ET_DiagExt.InitSubModulesException;
stInitSubModulesException.sDiagExt											:= FC_EtDiagExtToString(i_etDiagExt := stInitSubModulesException.udiDiagExt);
stInitSubModulesException.sMsg												:= '';	(* Replaced on usage *)
stInitSubModulesException.udiModuleId										:= iq_stStandardModuleItf.i_udiModuleId;
stInitSubModulesException.sModuleName										:= iq_stStandardModuleItf.i_sModuleName;
stInitSubModulesException.stReaction.axReaction[TPL.ET_Reaction.AsyncStop]	:= TRUE;
stInitSubModulesException.etSource											:= TPL.ET_ExceptionSource.NodeModule;
stInitSubModulesException.timDelayTime										:= T#0MS;
stInitSubModulesException.wHmiAttributes									:= 0;
stInitSubModulesException.xAutoQuit											:= FALSE;


(*------------------------------------------------------------------------------------------*)
(* Init User Exceptions *)

	// TPL.ET_Reaction.AsyncStop
	// TPL.ET_Reaction.SyncStopEL
	// TPL.ET_Reaction.SyncStopEH
	// TPL.ET_Reaction.StopEndOfCycle
	// TPL.ET_Reaction.MainsContactorOff

(*------------------------------------------------------------------------------------------*)
stUserException1.etDiag													:= GD.ET_Diag.ExecutionAborted;
stUserException1.udiDiagExt												:= ET_DiagExtUser.Exception1FromEquipmentModule;
stUserException1.sDiagExt												:= FC_EtDiagExtUserToString(i_etDiagExt := stUserException1.udiDiagExt);
stUserException1.sMsg													:= 'User Exception 1';
stUserException1.udiModuleId											:= iq_stStandardModuleItf.i_udiModuleId;
stUserException1.sModuleName											:= iq_stStandardModuleItf.i_sModuleName;
stUserException1.stReaction.axReaction[TPL.Gc_udiUserReactionOffset+2]	:= TRUE;
stUserException1.etSource												:= TPL.ET_ExceptionSource.User;
stUserException1.timDelayTime											:= T#0MS;
stUserException1.wHmiAttributes											:= 0;
stUserException1.xAutoQuit												:= FALSE;

stUserException2.etDiag													:= GD.ET_Diag.ExecutionAborted;
stUserException2.udiDiagExt												:= ET_DiagExtUser.Exception2FromEquipmentModule;
stUserException2.sDiagExt												:= FC_EtDiagExtUserToString(i_etDiagExt := stUserException2.udiDiagExt);
stUserException2.sMsg													:= 'User Exception 2';
stUserException2.udiModuleId											:= iq_stStandardModuleItf.i_udiModuleId;
stUserException2.sModuleName											:= iq_stStandardModuleItf.i_sModuleName;
stUserException2.stReaction.axReaction[TPL.Gc_udiUserReactionOffset+2]	:= TRUE;
stUserException2.etSource												:= TPL.ET_ExceptionSource.User;
stUserException2.timDelayTime											:= T#0MS;
stUserException2.wHmiAttributes											:= 0;
stUserException2.xAutoQuit												:= FALSE;

(* End of system generated code, could be modified for your application *)
END_ACTION

ACTION Init_Nocke1:
(* Standard interface *)
astSubModuleInterface[c_udiNocke1].i_sModuleName		:= CONCAT(STR1 := iq_stStandardModuleItf.i_sModuleName, STR2 := ': Nocke1');

astSubModuleInterface[c_udiNocke1].i_xLogEnable			:= TRUE;
astSubModuleInterface[c_udiNocke1].i_wLogDataFilter		:= UDINT_TO_WORD(TPL.ET_LogDataFilter.ModuleDefault);

(* ExampleLeafModule specific interface *)
stNocke1Interface.i_ifDrive				:= DRV_Master;
stNocke1Interface.i_lrPosMin			:= 120.0;
stNocke1Interface.i_lrPosMax			:= 250.0;
stNocke1Interface.i_xInitHoming			:= TRUE;
END_ACTION

ACTION Init_Reactions:
(* System generated code, only to be changed by experienced programmers *)
IF c_udiNumberOfSubModules < 1 THEN
	RETURN;
END_IF

(* Change of default reactions only on demand *)
(* Compare SR MainMachine Action Init_Reactions *)

xInitReactionsException := FALSE;

(*****************************************************************************************************************************************************)
(* Init ReactionTranslationMode *)

TPL.FC_InitReactionTranslationMode(	i_udiNumberOfSubModules			:= c_udiNumberOfSubModules,
									i_petReactionTranslationMode	:= ADR(aetReactionTranslationMode),
									q_etDiag						=> etDiag,
									q_etDiagExt						=> etDiagExtTPL);
							
IF etDiag <> GD.ET_Diag.Ok AND NOT xInitReactionsException THEN
	xInitReactionsException := TRUE;
	
	stInitReactionsException.sMsg := PDL.FC_MultiConcat(i_sString1 := 'InitReactionTranslationMode - ', 
														i_sString2 := GD.FC_EtDiagToString(i_etDiag := etDiag), 
														i_sString3 := ' - ', 
														i_sString4 := TPL.FC_EtDiagExtToString(i_etDiagExt := etDiagExtTPL));
END_IF	

(*****************************************************************************************************************************************************)
(* Init ReactionTranslationTable *)	

TPL.FC_InitReactionTranslationTable(i_udiNumberOfSubModules			:= c_udiNumberOfSubModules,
									i_pstReactionTranslationTable	:= ADR(aastReactionTranslationTable),
									q_etDiag						=> etDiag,
									q_etDiagExt						=> etDiagExtTPL);
									
IF etDiag <> GD.ET_Diag.Ok AND NOT xInitReactionsException THEN
	xInitReactionsException := TRUE;
	
	stInitReactionsException.sMsg := PDL.FC_MultiConcat(i_sString1 := 'InitReactionTranslationTable - ', 
														i_sString2 := GD.FC_EtDiagToString(i_etDiag := etDiag), 
														i_sString3 := ' - ', 
														i_sString4 := TPL.FC_EtDiagExtToString(i_etDiagExt := etDiagExtTPL));
END_IF		

(*****************************************************************************************************************************************************)
(* Init ReactionTranslationJobs *)	
								
TPL.FC_InitReactionTranslationJobs( i_udiNumberOfSubModules			:= c_udiNumberOfSubModules,
									i_pstReactionTranslationJobs	:= ADR(astReactionTranslationJobs),
									q_etDiag						=> etDiag,
									q_etDiagExt						=> etDiagExtTPL);
						
IF etDiag <> GD.ET_Diag.Ok AND NOT xInitReactionsException THEN
	xInitReactionsException := TRUE;
	
	stInitReactionsException.sMsg := PDL.FC_MultiConcat(i_sString1 := 'InitReactionTranslationJobs - ', 
														i_sString2 := GD.FC_EtDiagToString(i_etDiag := etDiag), 
														i_sString3 := ' - ', 
														i_sString4 := TPL.FC_EtDiagExtToString(i_etDiagExt := etDiagExtTPL));
END_IF		

(*****************************************************************************************************************************************************)
(* Set exception if any exception occurred *)

TPL.FC_SetException(i_xExceptionActive	:= xInitReactionsException, 
					iq_stException		:= stInitReactionsException, 
					iq_stExceptionList	:= iq_stExceptionList, 
					iq_stLogDataList	:= iq_stLogDataList);
					
xInitSuccessful := xInitSuccessful AND NOT xInitReactionsException;

etDiag := GD.ET_Diag.Ok;
(* End of system generated code, only to be changed by experienced programmers *)
END_ACTION

ACTION Init_Slave3:
(* System generated code, could be modified for your application *)

(* Standard interface *)
astSubModuleInterface[c_udiSlave3].i_sModuleName		:= CONCAT(STR1 := iq_stStandardModuleItf.i_sModuleName, STR2 := ': Slave3');

astSubModuleInterface[c_udiSlave3].i_xLogEnable			:= 	TRUE;
astSubModuleInterface[c_udiSlave3].i_wLogDataFilter		:= 	UDINT_TO_WORD(TPL.ET_LogDataFilter.ModuleDefault);

(* MotionModule specific interface *)
stSlave3Interface.stMain.i_ifMaster			:= i_ifMaster; 		(* Master *)
stSlave3Interface.stMain.i_ifDrive			:= DRV_Slave3;
stSlave3Interface.stMain.iq_lencEncoder		:= LE_Slave3;


xDriveIsVirtual := FC_IsDriveVirtual(	i_ifDrive	:= stSlave3Interface.stMain.i_ifDrive,
										q_etDiag	=> etDiag,
										q_etDiagExt	=> etDiagExt, //etDiagExtTPL,
										q_sMsg		=> sMsgBuffer);

IF etDiag <> GD.ET_Diag.Ok AND NOT xIsDriveVirtualException THEN										
	stIsDriveVirtualException.sMsg := sMsgBuffer;
	xIsDriveVirtualException := TRUE;
END_IF

TPL.FC_SetException(i_xExceptionActive	:= xIsDriveVirtualException, 
					iq_stException		:= stIsDriveVirtualException, 
					iq_stExceptionList	:= iq_stExceptionList, 
					iq_stLogDataList	:= iq_stLogDataList);
					
xInitSuccessful := xInitSuccessful AND NOT xIsDriveVirtualException;
etDiag := GD.ET_Diag.Ok;
	

(*Set DeadTime compensation parameters depending on used type of Master*)
FC_SetDeadTimeCompensation(i_stSubModuleInterfaceMain := stSlave3Interface.stMain);
  (*Please note, FC_DeadTimeCompensation does not recognize the master type, transferred via C2C or encoder network! 
	stXXXXInterface.stMain.iq_lencEncoder.Delay must be adjusted in order to reach shaft synchronism, it depends on:
	- Transmission delay via the choosen network, depending on topology and timing 
	- Type of the master e.g. physical encoder or an axis
	- SERCOS cycle times in master and slave controllers
	
	C2C sample (similar for encoder network):
	//Access C2C_EncIn.DataDelay only if C2C_Master.SyncGroupState=5 or C2C_Slave.SyncGroupState = 5 and C2C_EncIn.DataValid = TRUE!

		//Master is a physical encoder (PMEnc/Inc):
			stXXXXInterface.stMain.iq_lencEncoder.Delay := C2C_EncIn.DataDelay - DRV_SlaveAxis.ShaftRefDelay;

		//Master is an axis (real/ virtual):
			stXXXXInterface.stMain.iq_lencEncoder.Delay := C2C_EncIn.DataDelay + one SERCOS cycle of C2C controller with connected master axis;*)


stSlave3Interface.stMain.i_lrMotionActiveVelLimit						:= 15.0;	(* Limit for max. velocity of astAxisModuleInterface to switch output AxisMove in Units/s *)
stSlave3Interface.stMain.i_etMotionActiveVelType						:= AXM.ET_MotionActiveVelType.Velocity;

stSlave3Interface.stMain.i_timMasterStop								:= T#1S;
stSlave3Interface.stMain.i_xHwLimitPos									:= FALSE;
stSlave3Interface.stMain.i_xHwLimitNeg									:= FALSE;

stSlave3Interface.stMain.stReducedVelocity.i_xEnableReducedVelocity		:= FALSE;
stSlave3Interface.stMain.stReducedVelocity.i_xOnlyLimitCheck			:= FALSE;
stSlave3Interface.stMain.stReducedVelocity.i_lrMaxReducedVelocity		:= 50.0;

stSlave3Interface.stMain.i_xStart										:= FALSE;

(***************************************************************************************************************************************************************************************************)

(*** Homing ***)

IF xDriveIsVirtual THEN
	stSlave3Interface.stHome.i_etMode := PDL.ET_HomeMode.SetPosAxisAndLogEncoderPosition;			(* Homing Mode  in case of virtual axis *)
ELSE
	stSlave3Interface.stHome.i_etMode := PDL.ET_HomeMode.PosDirectionPosEdgeTp;						(* Homing Mode in case of real axis *)
END_IF


stSlave3Interface.stHome.i_xEnableInitAbsReadPos := FALSE;		(* TRUE : Restores the AxisPosition depending on the stHome.etMode
																		  If stHome.i_etMode is equal to PDL.ET_HomeMode.RestorePosFromAxisEncoder or 
																		  to PDL.ET_HomeMode.WriteAxisEncoder, the encoder of the axis is read,
																		  or else the position will be restored from the retain area *)
						   
stSlave3Interface.stHome.stSetpos.iq_pstRestorePosRetain := ADR(Grp_stRestorePositionAxis4);

stSlave3Interface.stHome.i_xResetHomeOk := FALSE;

(* Possible modes for homing mode Sensor:
	PDL.ET_HomeMode.PosDirectionPosEdgeSensor
	PDL.ET_HomeMode.NegDirectionPosEdgeSensor
	PDL.ET_HomeMode.NegDirectionNegEdgeSensor
	PDL.ET_HomeMode.PosDirectionNegEdgeSensor
*)
stSlave3Interface.stHome.stSensor.i_lrHomePosition			:= 0.0;			(* Position at the end of homing in units *)
stSlave3Interface.stHome.stSensor.i_lrVel					:= 10.0;		(* Homing ceiling velocity in units/s *)
stSlave3Interface.stHome.stSensor.i_lrAcc					:= 1000.0;		(* Homing acceleration in units/s^2 *)
stSlave3Interface.stHome.stSensor.i_lrDec					:= 1000.0;		(* Homing deceleration in units/s^2 *)
stSlave3Interface.stHome.stSensor.i_lrJerk					:= 10000.0;		(* Homing jerk in units/s^3 *)
stSlave3Interface.stHome.stSensor.i_lrOffset				:= 0.0;			(* Offset from home signal in units *)
stSlave3Interface.stHome.stSensor.i_lrMaxTravel				:= 720.0;		(* Max. travel for referencing by normal input *)
stSlave3Interface.stHome.stSensor.i_xRotativeSystem			:= FALSE;		(* Rotative system true or false for referencing by normal input *)
stSlave3Interface.stHome.stSensor.i_xSensor					:= FALSE;		(* Input for home signal. Can be a signal from a controller input. Has to be written cyclic. *)

(* Possible Modes for homing mode LimitSwitch:
	PDL.ET_HomeMode.PosDirectionPosEdgeHWLimitPos		normally open contact / Closing contact
	PDL.ET_HomeMode.NegDirectionPosEdgeHWLimitNeg		normally open contact / Closing contact
	PDL.ET_HomeMode.NegDirectionNegEdgeHWLimitNeg		normally closed contact / Opening contact  
	PDL.ET_HomeMode.PosDirectionNegEdgeHWLimitPos		normally closed contact / Opening contact 
*)
stSlave3Interface.stHome.stLimitSwitch.i_lrHomePosition		:= 0.0;			(* Position at the end of homing in units *)
stSlave3Interface.stHome.stLimitSwitch.i_lrVel				:= 10.0;		(* Homing ceiling velocity in units/s *)
stSlave3Interface.stHome.stLimitSwitch.i_lrLowVel			:= 5.0;			(* Homing low ceiling velocity in units/s *)
stSlave3Interface.stHome.stLimitSwitch.i_lrAcc				:= 1000.0;		(* Homing acceleration in units/s^2 *)
stSlave3Interface.stHome.stLimitSwitch.i_lrDec				:= 1000.0;		(* Homing deceleration in units/s^2 *)
stSlave3Interface.stHome.stLimitSwitch.i_lrJerk				:= 10000.0;		(* Homing jerk in units/s^3 *)
stSlave3Interface.stHome.stLimitSwitch.i_lrOffset			:= 0.0;			(* Offset from home signal in units *)
stSlave3Interface.stHome.stLimitSwitch.i_lrMaxTravel		:= 9999.0;		(* Max. travel for referencing normal input as a hardware limit *)

(* Possible modes for homing mode MoveOnPos:
	PDL.ET_HomeMode.MoveOnPosAbs 
*)
stSlave3Interface.stHome.stMoveonPos.i_lrTarget				:= 0.0;			(* Position at the end of homing in units *)
stSlave3Interface.stHome.stMoveonPos.i_lrVel				:= 10.0;		(* Homing ceiling velocity in units/s *)
stSlave3Interface.stHome.stMoveonPos.i_lrAcc				:= 1000.0;		(* Homing acceleration in units/s^2 *)
stSlave3Interface.stHome.stMoveonPos.i_lrDec				:= 1000.0;		(* Homing deceleration in units/s^2 *)
stSlave3Interface.stHome.stMoveonPos.i_lrJerk				:= 10000.0;		(* Homing jerk in units/s^3 *)
stSlave3Interface.stHome.stMoveonPos.i_lrPeriod				:= 0.0;			(* Period of the axis *)
stSlave3Interface.stHome.stMoveonPos.i_xRotativeSystem		:= FALSE;		(* Rotative system true or false *)

(* Possible modes for homing mode SetPos:
	PDL.ET_HomeMode.SetPosAxisPosition 
	PDL.ET_HomeMode.SetPosLogEncoderPosition 
	PDL.ET_HomeMode.SetPosAxisAndLogEncoderPosition
	PDL.ET_HomeMode.RestorePosFromAxisEncoder 
	PDL.ET_HomeMode.RestorePosFromRetain 
*)
stSlave3Interface.stHome.stSetpos.i_lrHomePosition			:= 0.0;			(* Position at the end of homing in units *)
stSlave3Interface.stHome.stSetpos.i_lrEncoderPosition		:= 0.0;			(* Encoder position in units after homing *)
stSlave3Interface.stHome.stSetpos.i_lrAbsEncOffset			:= 100.0;		(* Distance to the jump of axis encoder in units  *)
stSlave3Interface.stHome.stSetpos.i_lrRestoreWindow			:= 180;			(* How far can the drive be away from is correct position *)
stSlave3Interface.stHome.stSetpos.i_lrUserPeriod			:= 360;			(* Period of the axis *)

(* Possible modes for homing mode Torque:
	PDL.ET_HomeMode.PosDirectionMaxTorque 
	PDL.ET_HomeMode.NegDirectionMaxTorque 
*)
stSlave3Interface.stHome.stTorque.i_lrHomePosition			:= 0.0;			(* Position at the end of homing in units *)
stSlave3Interface.stHome.stTorque.i_lrVel					:= 10.0;		(* Homing ceiling velocity in units/s *)
stSlave3Interface.stHome.stTorque.i_lrAcc					:= 1000.0;		(* Homing acceleration in units/s^2 *)
stSlave3Interface.stHome.stTorque.i_lrDec					:= 1000.0;		(* Homing deceleration in units/s^2 *)
stSlave3Interface.stHome.stTorque.i_lrJerk					:= 10000.0;		(* Homing jerk in units/s^3 *)
stSlave3Interface.stHome.stTorque.i_lrOffset				:= 0.0;			(* Offset from home signal in units *)
stSlave3Interface.stHome.stTorque.i_lrMaxTravel				:= 9999.0;		(* Max. travel for referencing by torque *)
stSlave3Interface.stHome.stTorque.i_lrMaxTorque				:= 0.0;			(* Torque for stop in Nm / referencing by torque *)
stSlave3Interface.stHome.stTorque.i_diTorqueTime			:= 5;			(* Time in msec to hold torque *)

(* Possible modes for homing mode TouchProbe:
	PDL.ET_HomeMode.PosDirectionPosEdgeTp 
	PDL.ET_HomeMode.NegDirectionPosEdgeTp 
	PDL.ET_HomeMode.NegDirectionNegEdgeTp 
	PDL.ET_HomeMode.PosDirectionNegEdgeTp 
*)
stSlave3Interface.stHome.stTouchProbe.i_lrHomePosition		:= 0.0;			(* Position at the end of homing in units *)
stSlave3Interface.stHome.stTouchProbe.i_lrVel				:= 100.0;		(* Homing ceiling velocity in units/s *)
stSlave3Interface.stHome.stTouchProbe.i_lrAcc				:= 1000.0;		(* Homing acceleration in units/s^2 *)
stSlave3Interface.stHome.stTouchProbe.i_lrDec				:= 1000.0;		(* Homing deceleration in units/s^2 *)
stSlave3Interface.stHome.stTouchProbe.i_lrJerk				:= 10000.0;		(* Homing jerk in units/s^3 *)
stSlave3Interface.stHome.stTouchProbe.i_lrOffset			:= 30.0;		(* Offset from home signal in units *)
stSlave3Interface.stHome.stTouchProbe.i_lrMaxTravel			:= 720.0;		(* Max. travel for referencing by TP *)
stSlave3Interface.stHome.stTouchProbe.i_xRotativeSystem		:= TRUE;		(* Rotative system true or false for referencing by TP *)
stSlave3Interface.stHome.stTouchProbe.i_ifTouchProbe		:= TP_3;		(* Input for TP *)

(* Possible modes for homing mode WritePos:
	PDL.ET_HomeMode.WriteAxisEncoder 
*)
stSlave3Interface.stHome.stWritePos.i_lrHomePosition		:= 0.0;			(* Position at the end of homing in units *)
stSlave3Interface.stHome.stWritePos.i_lrUserPeriod			:= 0.0;			(* Calculates Drive.position into period ( units ) *)
stSlave3Interface.stHome.stWritePos.i_lrAbsEncOffset		:= 100.0;		(* Distance to the jump of axis encoder in units *)

(***************************************************************************************************************************************************************************************************)
(*** Manual ***)

stSlave3Interface.stManual.i_lrVel								:= 50.0;			(* Velocity in units/s *)
stSlave3Interface.stManual.i_lrAcc								:= 100.0;			(* Acceleration in units/s^2 *)
stSlave3Interface.stManual.i_lrDec								:= 100.0;			(* Deceleration in units/s^2 *)
stSlave3Interface.stManual.i_lrJerk								:= 1000.0;			(* Jerk in units/s^3 *)
stSlave3Interface.stManual.i_lrMaxDistance						:= 120.0;			(* Max pathlengths for one step in units *)
stSlave3Interface.stManual.i_xEndless							:= FALSE;			(* TRUE: jogging endless; Position between the periode; FALSE: jogging in steps. Position can be out of periode *)
stSlave3Interface.stManual.i_lrPeriod							:= 360.0;			(* Period of the axis *)

(***************************************************************************************************************************************************************************************************)
(*** Cam ***)

stSlave3Interface.stMultiCam.i_etCSModeSlave					:= PDL.ET_MultiCamCsModeSlave.SetSlavePositionToFirstCamPosition;		(* ColdStartMode Slave *)
stSlave3Interface.stMultiCam.i_etCSModeMaster					:= PDL.ET_MultiCamCsModeMaster.SetMasterPositionToFirstCamPosition;		(* ColdStartMode Master *)
stSlave3Interface.stMultiCam.i_etWSMode							:= PDL.ET_MultiCamWsMode.StoredCamMoveAlwaysNoPositionCheck;			(* WarmStartMode *)
stSlave3Interface.stMultiCam.i_lrWSWindow						:= 5.0;											(* WarmStartWindow in Axis units *)
stSlave3Interface.stMultiCam.i_lrWSVel							:= 10.0;										(* Velocity for WarmStart and CSModeSlave = PDL.ET_MultiCamCsModeSlave.MoveSlaveToFirstCamPosition in Units/s *)
stSlave3Interface.stMultiCam.i_lrWSAcc							:= 1000.0;										(* Acceleration and deceleration for Warmstart and CSModeSlave = PDL.ET_MultiCamCsModeSlave.MoveSlaveToFirstCamPosition in Units/s^2 *)
stSlave3Interface.stMultiCam.i_lrWSJerk							:= 10000.0;										(* Jerk for Warmstart and CSModeSlave = PDL.ET_MultiCamCsModeSlave.MoveSlaveToFirstCamPosition in units/s^3 *)
stSlave3Interface.stMultiCam.i_diTXend							:= 2*SYSTEMINTERFACE.FC_LzsTaskGetInterval();	(* Time of XLowEnd and XHighEnd befor Xend or Xstart in msec*)
stSlave3Interface.stMultiCam.i_lrInstantXLimMax					:= 0.0;											(* Switch off position at 'InstantNewCam' *)

stSlave3Interface.stMultiCam.i_xEnableTabHandler				:= TRUE;										(* TRUE: TabHandler is enabled *)
stSlave3Interface.stMultiCam.i_udiTableSelectNr					:= AXM.ET_ParId.User;							(* Number of table which is used in the next cycle *)								

stSlave3Interface.stMultiCam.i_xSetEncoderParameters			:= FALSE;										(* TRUE: The parameters MasterId, FeedConstand, GearIn and GearOut will be copyed into LEnc object *)
stSlave3Interface.stMultiCam.i_xSetEncoderPosition				:= FALSE;										(* TRUE: Manipulation of LEnc object on startup OpMode MultiCam *)
stSlave3Interface.stMultiCam.i_lrSetEncoderOffset				:= 0.0;											(* Master encoder offset *)
stSlave3Interface.stMultiCam.i_xCheckEncoderPeriod				:= TRUE;										(* TRUE: Check of encoder period = 0. If encoder period <> 0 -> Exception *)

stSlave3Interface.stMultiCam.iq_astMotionPar[AXM.ET_ParId.User].diNumberOfCamPoints		:= 4;	(* DataStruct for the next cycle *)
stSlave3Interface.stMultiCam.iq_astMotionPar[AXM.ET_ParId.User].lrYPeriod				:= 0.0;

stSlave3Interface.stMultiCam.iq_astMotionPar[AXM.ET_ParId.User].astCamPoint[0].lrX		:= 0.0;
stSlave3Interface.stMultiCam.iq_astMotionPar[AXM.ET_ParId.User].astCamPoint[0].lrY		:= 0.0;
stSlave3Interface.stMultiCam.iq_astMotionPar[AXM.ET_ParId.User].astCamPoint[0].lrM		:= 0.0;
stSlave3Interface.stMultiCam.iq_astMotionPar[AXM.ET_ParId.User].astCamPoint[0].etCamType	:= PDL.ET_CamType.Poly5Com;
stSlave3Interface.stMultiCam.iq_astMotionPar[AXM.ET_ParId.User].astCamPoint[1].lrX		:= 60.0;
stSlave3Interface.stMultiCam.iq_astMotionPar[AXM.ET_ParId.User].astCamPoint[1].lrY		:= 30.0;
stSlave3Interface.stMultiCam.iq_astMotionPar[AXM.ET_ParId.User].astCamPoint[1].lrM		:= 1.0;
stSlave3Interface.stMultiCam.iq_astMotionPar[AXM.ET_ParId.User].astCamPoint[1].etCamType	:= PDL.ET_CamType.Straight;
stSlave3Interface.stMultiCam.iq_astMotionPar[AXM.ET_ParId.User].astCamPoint[2].lrX		:= 240.0;
stSlave3Interface.stMultiCam.iq_astMotionPar[AXM.ET_ParId.User].astCamPoint[2].lrY		:= 210.0;
stSlave3Interface.stMultiCam.iq_astMotionPar[AXM.ET_ParId.User].astCamPoint[2].lrM		:= 1.0;
stSlave3Interface.stMultiCam.iq_astMotionPar[AXM.ET_ParId.User].astCamPoint[2].etCamType	:= PDL.ET_CamType.Poly5Com;
stSlave3Interface.stMultiCam.iq_astMotionPar[AXM.ET_ParId.User].astCamPoint[3].lrX		:= 360.0;
stSlave3Interface.stMultiCam.iq_astMotionPar[AXM.ET_ParId.User].astCamPoint[3].lrY		:= 0.0;
stSlave3Interface.stMultiCam.iq_astMotionPar[AXM.ET_ParId.User].astCamPoint[3].lrM		:= 0.0;
stSlave3Interface.stMultiCam.iq_astMotionPar[AXM.ET_ParId.User].astCamPoint[3].etCamType	:= PDL.ET_CamType.Poly5Com;

stSlave3Interface.stMultiCam.iq_astMotionPar[AXM.ET_ParId.Idle].diUserTableId	:= UDINT_TO_DINT(AXM.ET_ParId.Idle);
stSlave3Interface.stMultiCam.iq_astMotionPar[AXM.ET_ParId.Start].diUserTableId	:= UDINT_TO_DINT(AXM.ET_ParId.Start);
stSlave3Interface.stMultiCam.iq_astMotionPar[AXM.ET_ParId.Cont].diUserTableId	:= UDINT_TO_DINT(AXM.ET_ParId.Cont);
stSlave3Interface.stMultiCam.iq_astMotionPar[AXM.ET_ParId.Stop].diUserTableId	:= UDINT_TO_DINT(AXM.ET_ParId.Stop);
stSlave3Interface.stMultiCam.iq_astMotionPar[AXM.ET_ParId.User].diUserTableId	:= UDINT_TO_DINT(AXM.ET_ParId.User);


(***************************************************************************************************************************************************************************************************)
(*** Endless ***)

stSlave3Interface.stEndless.i_lrVel					:= 100.0;			(* Velocity in Units/s *)
stSlave3Interface.stEndless.i_lrAcc					:= 1000.0;			(* Acceleration in Units/s^2 *)
stSlave3Interface.stEndless.i_lrDec					:= 1000.0;			(* Deceleration in Units/s^2 *)
stSlave3Interface.stEndless.i_lrJerk				:= 10000.0;			(* Jerk in units/s^3 *)
stSlave3Interface.stEndless.i_lrPeriod				:= 360.0;			(* Period one cycle in units *)
stSlave3Interface.stEndless.i_lrStopPosition		:= 0.5;				(* Stop position in units *)


(***************************************************************************************************************************************************************************************************)
(*** Pos ***)

stSlave3Interface.stPos.i_etPosMode								:= SYSTEMINTERFACE.ET_PosMode.Endless;		(* SYSTEMINTERFACE.ET_PosMode.Endless, SYSTEMINTERFACE.ET_PosMode.Relative, SYSTEMINTERFACE.ET_PosMode.Absolute *)
stSlave3Interface.stPos.i_lrTarget								:= 360.0;									(* Target position or distance in Units *)
stSlave3Interface.stPos.i_lrVel									:= 360.0;									(* Ceiling velocity in Units/s *)
stSlave3Interface.stPos.i_lrAcc									:= 3600.0;									(* Acceleration in Units/s^2 *)
stSlave3Interface.stPos.i_lrDec									:= 3600.0;									(* Deceleration in Units/s^2 *)
stSlave3Interface.stPos.i_lrJerk								:= 36000.0;									(* Jerk in units/s^3 *)

(* End of system generated code, could be modified for your application *)
END_ACTION

ACTION Init_Slave4:
(* System generated code, could be modified for your application *)

(* Standard interface *)
astSubModuleInterface[c_udiSlave4].i_sModuleName		:= CONCAT(STR1 := iq_stStandardModuleItf.i_sModuleName, STR2 := ': Slave4');

astSubModuleInterface[c_udiSlave4].i_xLogEnable			:= 	TRUE;
astSubModuleInterface[c_udiSlave4].i_wLogDataFilter		:= 	UDINT_TO_WORD(TPL.ET_LogDataFilter.ModuleDefault);

(* AxisModule specific interface *)
stSlave4Interface.stMain.i_ifMaster			:= i_ifMaster; 		(* Master *)
stSlave4Interface.stMain.i_ifDrive			:= DRV_Slave4;
stSlave4Interface.stMain.iq_lencEncoder		:= LE_Slave4;


xDriveIsVirtual := FC_IsDriveVirtual(	i_ifDrive	:= stSlave4Interface.stMain.i_ifDrive,
										q_etDiag	=> etDiag,
										q_etDiagExt	=> etDiagExt, //etDiagExtTPL,
										q_sMsg		=> sMsgBuffer);

IF etDiag <> GD.ET_Diag.Ok AND NOT xIsDriveVirtualException THEN										
	stIsDriveVirtualException.sMsg := sMsgBuffer;
	xIsDriveVirtualException := TRUE;
END_IF

TPL.FC_SetException(i_xExceptionActive	:= xIsDriveVirtualException, 
					iq_stException		:= stIsDriveVirtualException, 
					iq_stExceptionList	:= iq_stExceptionList, 
					iq_stLogDataList	:= iq_stLogDataList);
					
xInitSuccessful := xInitSuccessful AND NOT xIsDriveVirtualException;
etDiag := GD.ET_Diag.Ok;
	

(*Set DeadTime compensation parameters depending on used type of Master*)
FC_SetDeadTimeCompensation(i_stSubModuleInterfaceMain := stSlave4Interface.stMain);
  (*Please note, FC_DeadTimeCompensation does not recognize the master type, transferred via C2C or encoder network! 
	stXXXXInterface.stMain.iq_lencEncoder.Delay must be adjusted in order to reach shaft synchronism, it depends on:
	- Transmission delay via the choosen network, depending on topology and timing 
	- Type of the master e.g. physical encoder or an axis
	- SERCOS cycle times in master and slave controllers
	
	C2C sample (similar for encoder network):
	//Access C2C_EncIn.DataDelay only if C2C_Master.SyncGroupState=5 or C2C_Slave.SyncGroupState = 5 and C2C_EncIn.DataValid = TRUE!

		//Master is a physical encoder (PMEnc/Inc):
			stXXXXInterface.stMain.iq_lencEncoder.Delay := C2C_EncIn.DataDelay - DRV_SlaveAxis.ShaftRefDelay;

		//Master is an axis (real/ virtual):
			stXXXXInterface.stMain.iq_lencEncoder.Delay := C2C_EncIn.DataDelay + one SERCOS cycle of C2C controller with connected master axis;*)


xFirstCall := TRUE;		// Used in Logic_Action to start movement in first cycle when OpMode is AXM.ET_OpMode.Positioning

stSlave4Interface.stMain.i_lrMotionActiveVelLimit						:= 15.0;	(* Limit for max. velocity of astAxisModuleInterface to switch output AxisMove in Units/s *)
stSlave4Interface.stMain.i_etMotionActiveVelType						:= AXM.ET_MotionActiveVelType.Velocity;

stSlave4Interface.stMain.i_timMasterStop								:= T#1S;
stSlave4Interface.stMain.i_xHwLimitPos									:= FALSE;
stSlave4Interface.stMain.i_xHwLimitNeg									:= FALSE;

stSlave4Interface.stMain.stReducedVelocity.i_xEnableReducedVelocity		:= FALSE;
stSlave4Interface.stMain.stReducedVelocity.i_xOnlyLimitCheck			:= FALSE;
stSlave4Interface.stMain.stReducedVelocity.i_lrMaxReducedVelocity		:= 50.0;

stSlave4Interface.stMain.i_xStart										:= FALSE;

(***************************************************************************************************************************************************************************************************)

(*** Homing ***)

IF xDriveIsVirtual THEN
	stSlave4Interface.stHome.i_etMode := PDL.ET_HomeMode.SetPosAxisAndLogEncoderPosition;			(* Homing Mode  in case of virtual axis *)
ELSE
	stSlave4Interface.stHome.i_etMode := PDL.ET_HomeMode.PosDirectionPosEdgeTp;						(* Homing Mode in case of real axis *)
END_IF


stSlave4Interface.stHome.i_xEnableInitAbsReadPos := FALSE;		(* TRUE : Restores the AxisPosition depending on the stHome.etMode
																		  If stHome.i_etMode is equal to PDL.ET_HomeMode.RestorePosFromAxisEncoder or 
																		  to PDL.ET_HomeMode.WriteAxisEncoder, the encoder of the axis is read,
																		  or else the position will be restored from the retain area *)
						   
stSlave4Interface.stHome.stSetpos.iq_pstRestorePosRetain := ADR(Grp_stRestorePositionAxis5);

stSlave4Interface.stHome.i_xResetHomeOk := FALSE;

(* Possible modes for homing mode Sensor:
	PDL.ET_HomeMode.PosDirectionPosEdgeSensor
	PDL.ET_HomeMode.NegDirectionPosEdgeSensor
	PDL.ET_HomeMode.NegDirectionNegEdgeSensor
	PDL.ET_HomeMode.PosDirectionNegEdgeSensor
*)
stSlave4Interface.stHome.stSensor.i_lrHomePosition			:= 0.0;			(* Position at the end of homing in units *)
stSlave4Interface.stHome.stSensor.i_lrVel					:= 10.0;		(* Homing ceiling velocity in units/s *)
stSlave4Interface.stHome.stSensor.i_lrAcc					:= 1000.0;		(* Homing acceleration in units/s^2 *)
stSlave4Interface.stHome.stSensor.i_lrDec					:= 1000.0;		(* Homing deceleration in units/s^2 *)
stSlave4Interface.stHome.stSensor.i_lrJerk					:= 10000.0;		(* Homing jerk in units/s^3 *)
stSlave4Interface.stHome.stSensor.i_lrOffset				:= 0.0;			(* Offset from home signal in units *)
stSlave4Interface.stHome.stSensor.i_lrMaxTravel				:= 720.0;		(* Max. travel for referencing by normal input *)
stSlave4Interface.stHome.stSensor.i_xRotativeSystem			:= FALSE;		(* Rotative system true or false for referencing by normal input *)
stSlave4Interface.stHome.stSensor.i_xSensor					:= FALSE;		(* Input for home signal. Can be a signal from a controller input. Has to be written cyclic. *)

(* Possible Modes for homing mode LimitSwitch:
	PDL.ET_HomeMode.PosDirectionPosEdgeHWLimitPos		normally open contact / Closing contact
	PDL.ET_HomeMode.NegDirectionPosEdgeHWLimitNeg		normally open contact / Closing contact
	PDL.ET_HomeMode.NegDirectionNegEdgeHWLimitNeg		normally closed contact / Opening contact  
	PDL.ET_HomeMode.PosDirectionNegEdgeHWLimitPos		normally closed contact / Opening contact 
*)
stSlave4Interface.stHome.stLimitSwitch.i_lrHomePosition		:= 0.0;			(* Position at the end of homing in units *)
stSlave4Interface.stHome.stLimitSwitch.i_lrVel				:= 10.0;		(* Homing ceiling velocity in units/s *)
stSlave4Interface.stHome.stLimitSwitch.i_lrLowVel			:= 5.0;			(* Homing low ceiling velocity in units/s *)
stSlave4Interface.stHome.stLimitSwitch.i_lrAcc				:= 1000.0;		(* Homing acceleration in units/s^2 *)
stSlave4Interface.stHome.stLimitSwitch.i_lrDec				:= 1000.0;		(* Homing deceleration in units/s^2 *)
stSlave4Interface.stHome.stLimitSwitch.i_lrJerk				:= 10000.0;		(* Homing jerk in units/s^3 *)
stSlave4Interface.stHome.stLimitSwitch.i_lrOffset			:= 0.0;			(* Offset from home signal in units *)
stSlave4Interface.stHome.stLimitSwitch.i_lrMaxTravel		:= 9999.0;		(* Max. travel for referencing normal input as a hardware limit *)

(* Possible modes for homing mode MoveOnPos:
	PDL.ET_HomeMode.MoveOnPosAbs 
*)
stSlave4Interface.stHome.stMoveonPos.i_lrTarget				:= 0.0;			(* Position at the end of homing in units *)
stSlave4Interface.stHome.stMoveonPos.i_lrVel				:= 10.0;		(* Homing ceiling velocity in units/s *)
stSlave4Interface.stHome.stMoveonPos.i_lrAcc				:= 1000.0;		(* Homing acceleration in units/s^2 *)
stSlave4Interface.stHome.stMoveonPos.i_lrDec				:= 1000.0;		(* Homing deceleration in units/s^2 *)
stSlave4Interface.stHome.stMoveonPos.i_lrJerk				:= 10000.0;		(* Homing jerk in units/s^3 *)
stSlave4Interface.stHome.stMoveonPos.i_lrPeriod				:= 0.0;			(* Period of the axis *)
stSlave4Interface.stHome.stMoveonPos.i_xRotativeSystem		:= FALSE;		(* Rotative system true or false *)

(* Possible modes for homing mode SetPos:
	PDL.ET_HomeMode.SetPosAxisPosition 
	PDL.ET_HomeMode.SetPosLogEncoderPosition 
	PDL.ET_HomeMode.SetPosAxisAndLogEncoderPosition
	PDL.ET_HomeMode.RestorePosFromAxisEncoder 
	PDL.ET_HomeMode.RestorePosFromRetain 
*)
stSlave4Interface.stHome.stSetpos.i_lrHomePosition			:= 0.0;			(* Position at the end of homing in units *)
stSlave4Interface.stHome.stSetpos.i_lrEncoderPosition		:= 0.0;			(* Encoder position in units after homing *)
stSlave4Interface.stHome.stSetpos.i_lrAbsEncOffset			:= 100.0;		(* Distance to the jump of axis encoder in units  *)
stSlave4Interface.stHome.stSetpos.i_lrRestoreWindow			:= 180;			(* How far can the drive be away from is correct position *)
stSlave4Interface.stHome.stSetpos.i_lrUserPeriod			:= 360;			(* Period of the axis *)

(* Possible modes for homing mode Torque:
	PDL.ET_HomeMode.PosDirectionMaxTorque 
	PDL.ET_HomeMode.NegDirectionMaxTorque 
*)
stSlave4Interface.stHome.stTorque.i_lrHomePosition			:= 0.0;			(* Position at the end of homing in units *)
stSlave4Interface.stHome.stTorque.i_lrVel					:= 10.0;		(* Homing ceiling velocity in units/s *)
stSlave4Interface.stHome.stTorque.i_lrAcc					:= 1000.0;		(* Homing acceleration in units/s^2 *)
stSlave4Interface.stHome.stTorque.i_lrDec					:= 1000.0;		(* Homing deceleration in units/s^2 *)
stSlave4Interface.stHome.stTorque.i_lrJerk					:= 10000.0;		(* Homing jerk in units/s^3 *)
stSlave4Interface.stHome.stTorque.i_lrOffset				:= 0.0;			(* Offset from home signal in units *)
stSlave4Interface.stHome.stTorque.i_lrMaxTravel				:= 9999.0;		(* Max. travel for referencing by torque *)
stSlave4Interface.stHome.stTorque.i_lrMaxTorque				:= 0.0;			(* Torque for stop in Nm / referencing by torque *)
stSlave4Interface.stHome.stTorque.i_diTorqueTime			:= 5;			(* Time in msec to hold torque *)

(* Possible modes for homing mode TouchProbe:
	PDL.ET_HomeMode.PosDirectionPosEdgeTp 
	PDL.ET_HomeMode.NegDirectionPosEdgeTp 
	PDL.ET_HomeMode.NegDirectionNegEdgeTp 
	PDL.ET_HomeMode.PosDirectionNegEdgeTp 
*)
stSlave4Interface.stHome.stTouchProbe.i_lrHomePosition		:= 0.0;			(* Position at the end of homing in units *)
stSlave4Interface.stHome.stTouchProbe.i_lrVel				:= 100.0;		(* Homing ceiling velocity in units/s *)
stSlave4Interface.stHome.stTouchProbe.i_lrAcc				:= 1000.0;		(* Homing acceleration in units/s^2 *)
stSlave4Interface.stHome.stTouchProbe.i_lrDec				:= 1000.0;		(* Homing deceleration in units/s^2 *)
stSlave4Interface.stHome.stTouchProbe.i_lrJerk				:= 10000.0;		(* Homing jerk in units/s^3 *)
stSlave4Interface.stHome.stTouchProbe.i_lrOffset			:= 30.0;		(* Offset from home signal in units *)
stSlave4Interface.stHome.stTouchProbe.i_lrMaxTravel			:= 720.0;		(* Max. travel for referencing by TP *)
stSlave4Interface.stHome.stTouchProbe.i_xRotativeSystem		:= TRUE;		(* Rotative system true or false for referencing by TP *)
stSlave4Interface.stHome.stTouchProbe.i_ifTouchProbe		:= TP_4;		(* Input for TP *)

(* Possible modes for homing mode WritePos:
	PDL.ET_HomeMode.WriteAxisEncoder 
*)
stSlave4Interface.stHome.stWritePos.i_lrHomePosition		:= 0.0;			(* Position at the end of homing in units *)
stSlave4Interface.stHome.stWritePos.i_lrUserPeriod			:= 0.0;			(* Calculates Drive.position into period ( units ) *)
stSlave4Interface.stHome.stWritePos.i_lrAbsEncOffset		:= 100.0;		(* Distance to the jump of axis encoder in units *)

(***************************************************************************************************************************************************************************************************)
(*** Manual ***)

stSlave4Interface.stManual.i_lrVel								:= 50.0;			(* Velocity in units/s *)
stSlave4Interface.stManual.i_lrAcc								:= 100.0;			(* Acceleration in units/s^2 *)
stSlave4Interface.stManual.i_lrDec								:= 100.0;			(* Deceleration in units/s^2 *)
stSlave4Interface.stManual.i_lrJerk								:= 1000.0;			(* Jerk in units/s^3 *)
stSlave4Interface.stManual.i_lrMaxDistance						:= 120.0;			(* Max pathlengths for one step in units *)
stSlave4Interface.stManual.i_xEndless							:= FALSE;			(* TRUE: jogging endless; Position between the periode; FALSE: jogging in steps. Position can be out of periode *)
stSlave4Interface.stManual.i_lrPeriod							:= 360.0;			(* Period of the axis *)

(***************************************************************************************************************************************************************************************************)
(*** Cam ***)

stSlave4Interface.stMultiCam.i_etCSModeSlave					:= PDL.ET_MultiCamCsModeSlave.SetSlavePositionToFirstCamPosition;		(* ColdStartMode Slave *)
stSlave4Interface.stMultiCam.i_etCSModeMaster					:= PDL.ET_MultiCamCsModeMaster.SetMasterPositionToFirstCamPosition;		(* ColdStartMode Master *)
stSlave4Interface.stMultiCam.i_etWSMode							:= PDL.ET_MultiCamWsMode.StoredCamMoveAlwaysNoPositionCheck;			(* WarmStartMode *)
stSlave4Interface.stMultiCam.i_lrWSWindow						:= 5.0;											(* WarmStartWindow in Axis units *)
stSlave4Interface.stMultiCam.i_lrWSVel							:= 10.0;										(* Velocity for WarmStart and CSModeSlave = PDL.ET_MultiCamCsModeSlave.MoveSlaveToFirstCamPosition in Units/s *)
stSlave4Interface.stMultiCam.i_lrWSAcc							:= 1000.0;										(* Acceleration and deceleration for Warmstart and CSModeSlave = PDL.ET_MultiCamCsModeSlave.MoveSlaveToFirstCamPosition in Units/s^2 *)
stSlave4Interface.stMultiCam.i_lrWSJerk							:= 10000.0;										(* Jerk for Warmstart and CSModeSlave = PDL.ET_MultiCamCsModeSlave.MoveSlaveToFirstCamPosition in units/s^3 *)
stSlave4Interface.stMultiCam.i_diTXend							:= 2*SYSTEMINTERFACE.FC_LzsTaskGetInterval();	(* Time of XLowEnd and XHighEnd befor Xend or Xstart in msec*)
stSlave4Interface.stMultiCam.i_lrInstantXLimMax					:= 0.0;											(* Switch off position at 'InstantNewCam' *)

stSlave4Interface.stMultiCam.i_xEnableTabHandler				:= TRUE;										(* TRUE: TabHandler is enabled *)
stSlave4Interface.stMultiCam.i_udiTableSelectNr					:= AXM.ET_ParId.User;							(* Number of table which is used in the next cycle *)								

stSlave4Interface.stMultiCam.i_xSetEncoderParameters			:= FALSE;										(* TRUE: The parameters MasterId, FeedConstand, GearIn and GearOut will be copyed into LEnc object *)
stSlave4Interface.stMultiCam.i_xSetEncoderPosition				:= FALSE;										(* TRUE: Manipulation of LEnc object on startup OpMode MultiCam *)
stSlave4Interface.stMultiCam.i_lrSetEncoderOffset				:= 0.0;											(* Master encoder offset *)
stSlave4Interface.stMultiCam.i_xCheckEncoderPeriod				:= TRUE;										(* TRUE: Check of encoder period = 0. If encoder period <> 0 -> Exception *)

stSlave4Interface.stMultiCam.iq_astMotionPar[AXM.ET_ParId.User].diNumberOfCamPoints		:= 4;	(* DataStruct for the next cycle *)
stSlave4Interface.stMultiCam.iq_astMotionPar[AXM.ET_ParId.User].lrYPeriod				:= 0.0;

stSlave4Interface.stMultiCam.iq_astMotionPar[AXM.ET_ParId.User].astCamPoint[0].lrX		:= 0.0;
stSlave4Interface.stMultiCam.iq_astMotionPar[AXM.ET_ParId.User].astCamPoint[0].lrY		:= 0.0;
stSlave4Interface.stMultiCam.iq_astMotionPar[AXM.ET_ParId.User].astCamPoint[0].lrM		:= 0.0;
stSlave4Interface.stMultiCam.iq_astMotionPar[AXM.ET_ParId.User].astCamPoint[0].etCamType	:= PDL.ET_CamType.Poly5Com;
stSlave4Interface.stMultiCam.iq_astMotionPar[AXM.ET_ParId.User].astCamPoint[1].lrX		:= 60.0;
stSlave4Interface.stMultiCam.iq_astMotionPar[AXM.ET_ParId.User].astCamPoint[1].lrY		:= 30.0;
stSlave4Interface.stMultiCam.iq_astMotionPar[AXM.ET_ParId.User].astCamPoint[1].lrM		:= 1.0;
stSlave4Interface.stMultiCam.iq_astMotionPar[AXM.ET_ParId.User].astCamPoint[1].etCamType	:= PDL.ET_CamType.Straight;
stSlave4Interface.stMultiCam.iq_astMotionPar[AXM.ET_ParId.User].astCamPoint[2].lrX		:= 240.0;
stSlave4Interface.stMultiCam.iq_astMotionPar[AXM.ET_ParId.User].astCamPoint[2].lrY		:= 210.0;
stSlave4Interface.stMultiCam.iq_astMotionPar[AXM.ET_ParId.User].astCamPoint[2].lrM		:= 1.0;
stSlave4Interface.stMultiCam.iq_astMotionPar[AXM.ET_ParId.User].astCamPoint[2].etCamType	:= PDL.ET_CamType.Poly5Com;
stSlave4Interface.stMultiCam.iq_astMotionPar[AXM.ET_ParId.User].astCamPoint[3].lrX		:= 360.0;
stSlave4Interface.stMultiCam.iq_astMotionPar[AXM.ET_ParId.User].astCamPoint[3].lrY		:= 0.0;
stSlave4Interface.stMultiCam.iq_astMotionPar[AXM.ET_ParId.User].astCamPoint[3].lrM		:= 0.0;
stSlave4Interface.stMultiCam.iq_astMotionPar[AXM.ET_ParId.User].astCamPoint[3].etCamType	:= PDL.ET_CamType.Poly5Com;

stSlave4Interface.stMultiCam.iq_astMotionPar[AXM.ET_ParId.Idle].diUserTableId	:= UDINT_TO_DINT(AXM.ET_ParId.Idle);
stSlave4Interface.stMultiCam.iq_astMotionPar[AXM.ET_ParId.Start].diUserTableId	:= UDINT_TO_DINT(AXM.ET_ParId.Start);
stSlave4Interface.stMultiCam.iq_astMotionPar[AXM.ET_ParId.Cont].diUserTableId	:= UDINT_TO_DINT(AXM.ET_ParId.Cont);
stSlave4Interface.stMultiCam.iq_astMotionPar[AXM.ET_ParId.Stop].diUserTableId	:= UDINT_TO_DINT(AXM.ET_ParId.Stop);
stSlave4Interface.stMultiCam.iq_astMotionPar[AXM.ET_ParId.User].diUserTableId	:= UDINT_TO_DINT(AXM.ET_ParId.User);


(***************************************************************************************************************************************************************************************************)
(*** Endless ***)

stSlave4Interface.stEndless.i_lrVel								:= 100.0;			(* Velocity in Units/s *)
stSlave4Interface.stEndless.i_lrAcc								:= 1000.0;			(* Acceleration in Units/s^2 *)
stSlave4Interface.stEndless.i_lrDec								:= 1000.0;			(* Deceleration in Units/s^2 *)
stSlave4Interface.stEndless.i_lrJerk							:= 10000.0;			(* Jerk in units/s^3 *)
stSlave4Interface.stEndless.i_lrPeriod							:= 360.0;			(* Period one cycle in units *)
stSlave4Interface.stEndless.i_lrStopPosition					:= 0.5;				(* Stop position in units *)


(***************************************************************************************************************************************************************************************************)
(*** Pos ***)

stSlave4Interface.stPos.i_etPosMode								:= SYSTEMINTERFACE.ET_PosMode.Endless;		(* SYSTEMINTERFACE.ET_PosMode.Endless, SYSTEMINTERFACE.ET_PosMode.Relative, SYSTEMINTERFACE.ET_PosMode.Absolute *)
stSlave4Interface.stPos.i_lrTarget								:= 360.0;									(* Target position or distance in Units *)
stSlave4Interface.stPos.i_lrVel									:= 100.0;									(* Ceiling velocity in Units/s *)
stSlave4Interface.stPos.i_lrAcc									:= 3600.0;									(* Acceleration in Units/s^2 *)
stSlave4Interface.stPos.i_lrDec									:= 3600.0;									(* Deceleration in Units/s^2 *)
stSlave4Interface.stPos.i_lrJerk								:= 36000.0;									(* Jerk in units/s^3 *)

(* End of system generated code, could be modified for your application *)
END_ACTION

ACTION Init_SubModules:
(* System generated code, could be modified for your application *)

(*** Module Group declaration ***)

aaudiSubModuleGroups[c_udiCharlyGroup1-TPL.Gc_udiGroupOffset,TPL.ET_Group.Member1] := 0;				(* There is no first element of the group c_diCharlyGroup1 *)
aaudiSubModuleGroups[c_udiCharlyGroup1-TPL.Gc_udiGroupOffset,TPL.ET_Group.Member2] := 0;				(* There is no second element of the group c_diCharlyGroup1 *)

aaudiSubModuleGroups[c_udiCharlyGroup2-TPL.Gc_udiGroupOffset,TPL.ET_Group.Member1] := c_udiSlave3;	(* The Slave3 is the first element of the group c_diCharlyGroup2 *)
aaudiSubModuleGroups[c_udiCharlyGroup2-TPL.Gc_udiGroupOffset,TPL.ET_Group.Member2] := c_udiSlave4;	(* The Slave4 is the second element of the group c_diCharlyGroup2 *)

(* End of system generated code, could be modified for your application *)


(* System generated code, do not change without consulting 'Schneider Electric Automation GmbH' - otherwise you risk instability!!!*)
xInitSubModulesException := FALSE;

(*****************************************************************************************************************************************************)
(* Set IDs of SubModules *)	

TPL.FC_SetSubModuleIds(	i_udiMainModuleID			:= iq_stStandardModuleItf.i_udiModuleId,
						i_pstSubModulesItf			:= ADR(astSubModuleInterface),
						i_udiNumberOfSubModules		:= c_udiNumberOfSubModules,
						q_etDiag					=> etDiag,
						q_etDiagExt					=> etDiagExtTPL);
					
IF etDiag <> GD.ET_Diag.Ok AND NOT xInitSubModulesException THEN
	xInitSubModulesException := TRUE;
	
	stInitSubModulesException.sMsg := PDL.FC_MultiConcat(	i_sString1 := 'SetSubModuleIds - ', 
															i_sString2 := GD.FC_EtDiagToString(i_etDiag := etDiag), 
															i_sString3 := ' - ', 
															i_sString4 := TPL.FC_EtDiagExtToString(i_etDiagExt := etDiagExtTPL));
END_IF	

(*****************************************************************************************************************************************************)
(* Set exception if any exception occurred *)

TPL.FC_SetException(i_xExceptionActive	:= xInitSubModulesException, 
					iq_stException		:= stInitSubModulesException, 
					iq_stExceptionList	:= iq_stExceptionList, 
					iq_stLogDataList	:= iq_stLogDataList);

xInitSuccessful := xInitSuccessful AND NOT xInitSubModulesException;
					
etDiag := GD.ET_Diag.Ok;
(* End of system generated code, do not change without consulting 'Schneider Electric Automation GmbH' - otherwise you risk instability!!!*)
END_ACTION

ACTION InitModule_Action:
(* This step is used for initialisations after being enabled *)

(* System generated code, could be modified for your application *)
xInitSuccessful := TRUE;

Init_Exceptions();
(* End of system generated code, could be modified for your application *)

(* System generated code, do not change without consulting 'Schneider Electric Automation GmbH' - otherwise you risk instability!!!*)
iq_stStandardModuleItf.q_xActive			:= TRUE;
iq_stStandardModuleItf.q_xReady			:= FALSE;
iq_stStandardModuleItf.q_etDiag			:= GD.ET_Diag.Ok;
iq_stStandardModuleItf.q_udiDiagExt		:= ET_DiagExt.Initializing;
iq_stStandardModuleItf.q_sDiagExt			:= FC_EtDiagExtToString(i_etDiagExt := ET_DiagExt.Initializing);
iq_stStandardModuleItf.q_sMsg				:= '';

Init_SubModules();
Init_CmdTables();
Init_Reactions();
UpdateStructs();
(* End of system generated code, do not change without consulting 'Schneider Electric Automation GmbH' - otherwise you risk instability!!!*)

(* System generated code, could be modified for your application *)
Init_Slave3();
Init_Slave4();
Init_CrankModule(); (* calling CrankModule Initiation *)
Init_Nocke1();
(* End of system generated code, could be modified for your application *)

(* Application specific code *)
(* ToDo: Add your application specific code here *)
	;
(* End of application specific code *)
END_ACTION

ACTION Input_Action:
(* System generated code, do not change without consulting 'Schneider Electric Automation GmbH' - otherwise you risk instability!!!*)
UpdateStructs();
(* End of system generated code, do not change without consulting 'Schneider Electric Automation GmbH' - otherwise you risk instability!!!*)
END_ACTION

ACTION Logger_Action:
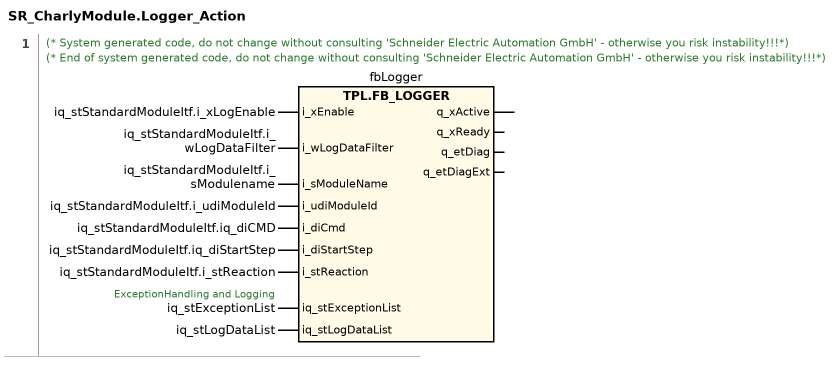
// NETWORK 1
// (* System generated code, do not change without consulting 'Schneider Electric Automation GmbH' - otherwise you risk instability!!!*)
// (* End of system generated code, do not change without consulting 'Schneider Electric Automation GmbH' - otherwise you risk instability!!!*)
//   fbLogger: Logging related variables
//   iq_stExceptionList: ExceptionHandling and Logging
fbLogger(
    i_xEnable := iq_stStandardModuleItf.i_xLogEnable,
    i_wLogDataFilter := iq_stStandardModuleItf.i_wLogDataFilter,
    i_sModuleName := iq_stStandardModuleItf.i_sModulename,
    i_udiModuleId := iq_stStandardModuleItf.i_udiModuleId,
    i_diCmd := iq_stStandardModuleItf.iq_diCMD,
    i_diStartStep := iq_stStandardModuleItf.iq_diStartStep,
    i_stReaction := iq_stStandardModuleItf.i_stReaction,
    iq_stExceptionList := iq_stExceptionList,
    iq_stLogDataList := iq_stLogDataList); // TPL.FB_LOGGER
END_ACTION

ACTION Logic_Action:
(* This is an example of how to use the Positioning mode *)

IF stSlave4Interface.stMain.q_etOpMode = AXM.ET_OpMode.Positioning THEN
	IF stSlave4Interface.stMain.q_xMotionActive THEN
		(* There must be a rising edge at the xStart bit for initializing new Pos values, therefore it have to be reset. *)
		 stSlave4Interface.stMain.i_xStart := FALSE;
	END_IF

	CASE iPosState OF
		1: (* moving back *)
			(* Wait until the InPosition signal *)
			IF stSlave4Interface.stPos.q_xInPosition THEN
				(*Initialize new Pos values*)
				stSlave4Interface.stPos.i_lrTarget	:= -360.0;
				stSlave4Interface.stPos.i_etPosMode	:= SYSTEMINTERFACE.ET_PosMode.Endless;
				
				iPosState := 2;
			END_IF
			
		2: (* moving forward *)
			(* Wait until the InPosition signal *)
			IF stSlave4Interface.stPos.q_xInPosition THEN
				(* Initialize new Pos values *)
				stSlave4Interface.stPos.i_lrTarget	:= 360.0;
				stSlave4Interface.stPos.i_etPosMode	:= SYSTEMINTERFACE.ET_PosMode.Endless;
				
				iPosState := 1;
			END_IF
	END_CASE
	
	(* Start movement again and set new initialized values *)
	IF xFirstCall THEN
		xFirstCall := FALSE;
		
		stSlave4Interface.stMain.i_xStart := TRUE;
		
	ELSIF NOT stSlave4Interface.stMain.q_xMotionActive AND stSlave4Interface.stPos.q_xInPosition THEN
		stSlave4Interface.stMain.i_xStart := TRUE;
	END_IF
ELSE
	(* Allows a re-start of the positioning movement after a Hold command *)
	xFirstCall := TRUE;

	(* Set the SYSTEMINTERFACE.ET_PosMode.Absolute mode that the movement will start later at the last position. *)
	stSlave4Interface.stPos.i_etPosMode := SYSTEMINTERFACE.ET_PosMode.Absolute;
	
	IF stSlave4Interface.stMain.q_etOpMode = AXM.ET_OpMode.Homing THEN
		(* Start with moving forward after homing *)
		stSlave4Interface.stPos.i_lrTarget := 360.0;
		
		iPosState := 1; (* next moving back *)
	END_IF
END_IF
END_ACTION

ACTION ModuleFaults:
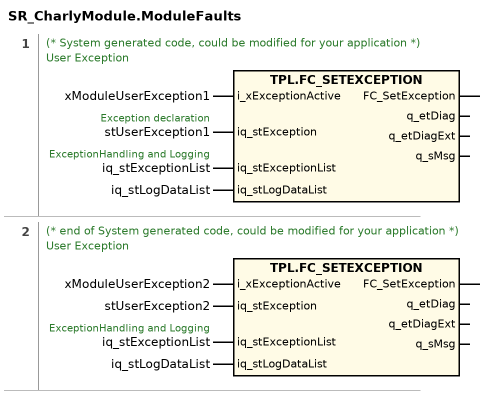
// NETWORK 1
// (* System generated code, could be modified for your application *)
// User Exception
//   stUserException1: Exception declaration
//   iq_stExceptionList: ExceptionHandling and Logging
TPL.FC_SETEXCEPTION(i_xExceptionActive := xModuleUserException1, iq_stException := stUserException1, iq_stExceptionList := iq_stExceptionList, iq_stLogDataList := iq_stLogDataList);

// NETWORK 2
// (* end of System generated code, could be modified for your application *)
// User Exception
//   iq_stExceptionList: ExceptionHandling and Logging
TPL.FC_SETEXCEPTION(i_xExceptionActive := xModuleUserException2, iq_stException := stUserException2, iq_stExceptionList := iq_stExceptionList, iq_stLogDataList := iq_stLogDataList);
END_ACTION

ACTION Output_Active:
(* System generated code, only to be changed by experienced programmers *)
IF iq_stStandardModuleItf.q_udiSubModuleInException <> 0 THEN
	iq_stStandardModuleItf.q_etDiag		:= GD.ET_Diag.Ok;
	iq_stStandardModuleItf.q_udiDiagExt	:= ET_DiagExt.SubModuleInException;
	iq_stStandardModuleItf.q_sDiagExt		:= FC_EtDiagExtToString(i_etDiagExt := ET_DiagExt.SubModuleInException);
	iq_stStandardModuleItf.q_sMsg			:= '';
ELSE
	IF etDiagModuleController = GD.ET_Diag.Ok THEN
		iq_stStandardModuleItf.q_etDiag	:= etDiagModuleController;
		iq_stStandardModuleItf.q_sMsg		:= sMsgModuleController;
		
		CASE etDiagExtModuleController OF
			TPL.ET_DiagExt.DeactivatingSubModules : 
				iq_stStandardModuleItf.q_udiDiagExt	:= ET_DiagExt.DeactivatingSubModules;
				iq_stStandardModuleItf.q_sDiagExt		:= FC_EtDiagExtToString(i_etDiagExt := ET_DiagExt.DeactivatingSubModules);
			TPL.ET_DiagExt.Disabled : 
				iq_stStandardModuleItf.q_udiDiagExt	:= ET_DiagExt.Disabled;
				iq_stStandardModuleItf.q_sDiagExt		:= FC_EtDiagExtToString(i_etDiagExt := ET_DiagExt.Disabled);
			TPL.ET_DiagExt.ExecuteStep : 
				iq_stStandardModuleItf.q_udiDiagExt	:= ET_DiagExt.ExecuteStep;
				iq_stStandardModuleItf.q_sDiagExt		:= FC_EtDiagExtToString(i_etDiagExt := ET_DiagExt.ExecuteStep);
			TPL.ET_DiagExt.Initializing : 
				iq_stStandardModuleItf.q_udiDiagExt	:= ET_DiagExt.Initializing;
				iq_stStandardModuleItf.q_sDiagExt		:= FC_EtDiagExtToString(i_etDiagExt := ET_DiagExt.Initializing);
			TPL.ET_DiagExt.WaitAtNegativeStep : 
				iq_stStandardModuleItf.q_udiDiagExt	:= ET_DiagExt.WaitAtNegativeStep;
				iq_stStandardModuleItf.q_sDiagExt		:= FC_EtDiagExtToString(i_etDiagExt := ET_DiagExt.WaitAtNegativeStep);
			TPL.ET_DiagExt.WaitCmdsDone : 
				iq_stStandardModuleItf.q_udiDiagExt	:= ET_DiagExt.WaitCmdsDone;
				iq_stStandardModuleItf.q_sDiagExt		:= FC_EtDiagExtToString(i_etDiagExt := ET_DiagExt.WaitCmdsDone);
			TPL.ET_DiagExt.WaitForCmd : 
				iq_stStandardModuleItf.q_udiDiagExt	:= ET_DiagExt.WaitForCmd;
				iq_stStandardModuleItf.q_sDiagExt		:= FC_EtDiagExtToString(i_etDiagExt := ET_DiagExt.WaitForCmd);
			ELSE
				iq_stStandardModuleItf.q_etDiag		:= GD. ET_Diag.UnexpectedProgramBehavior;
				iq_stStandardModuleItf.q_udiDiagExt	:= ET_DiagExt.UnknownStateModuleController;
				iq_stStandardModuleItf.q_sDiagExt		:= FC_EtDiagExtToString(i_etDiagExt := ET_DiagExt.UnknownStateModuleController);
		END_CASE
	ELSE
		iq_stStandardModuleItf.q_etDiag		:= GD.ET_Diag.DiagActive;
		iq_stStandardModuleItf.q_udiDiagExt	:= ET_DiagExt.ModuleControllerException;
		iq_stStandardModuleItf.q_sDiagExt		:= FC_EtDiagExtToString(i_etDiagExt := ET_DiagExt.ModuleControllerException);
		iq_stStandardModuleItf.q_sMsg			:= PDL.FC_MultiConcat(	i_sString1 := GD.FC_EtDiagToString(i_etDiag := etDiagModuleController), 
																			i_sString2 := ' - ',
																			i_sString3 := TPL.FC_EtDiagExtToString(i_etDiagExt := etDiagExtModuleController), 
																			i_sString4 := '');
	END_IF
END_IF

(* End of system generated code, only to be changed by experienced programmers *)
END_ACTION

ACTION Start_Action:
(* This step is active until the machine is being enabled *)

(* System generated code, do not change without consulting 'Schneider Electric Automation GmbH' - otherwise you risk instability!!! *)
iq_stStandardModuleItf.q_xActive			:= FALSE;
iq_stStandardModuleItf.q_xReady			:= FALSE;

iq_stStandardModuleItf.q_etDiag			:= GD.ET_Diag.Ok;
iq_stStandardModuleItf.q_udiDiagExt		:= ET_DiagExt.Disabled;
iq_stStandardModuleItf.q_sDiagExt			:= FC_EtDiagExtToString(i_etDiagExt := iq_stStandardModuleItf.q_udiDiagExt);
iq_stStandardModuleItf.q_sMsg				:= '';

iq_stStandardModuleItf.q_dwModuleType		:= TPL.ET_ModuleType.NodeModule;
iq_stStandardModuleItf.q_sModuleTypeName	:= 'NodeModule';
iq_stStandardModuleItf.q_udiModuleVersion	:= 1;	
(* End of system generated code, do not change without consulting 'Schneider Electric Automation GmbH' - otherwise you risk instability!!! *)

(* System generated code, to be changed by experienced programmers *)
IF iq_stStandardModuleItf.iq_diCMD <> 0 AND NOT iq_stStandardModuleItf.i_xEnable THEN
	iq_stStandardModuleItf.iq_diCMD := 0;
END_IF
(* End of system generated code, to be changed by experienced programmers *)

(* Application specific code *)
(* ToDo: Add your application specific code here *)
;
(* End of application specific code *)
END_ACTION

ACTION SubModules_Action:
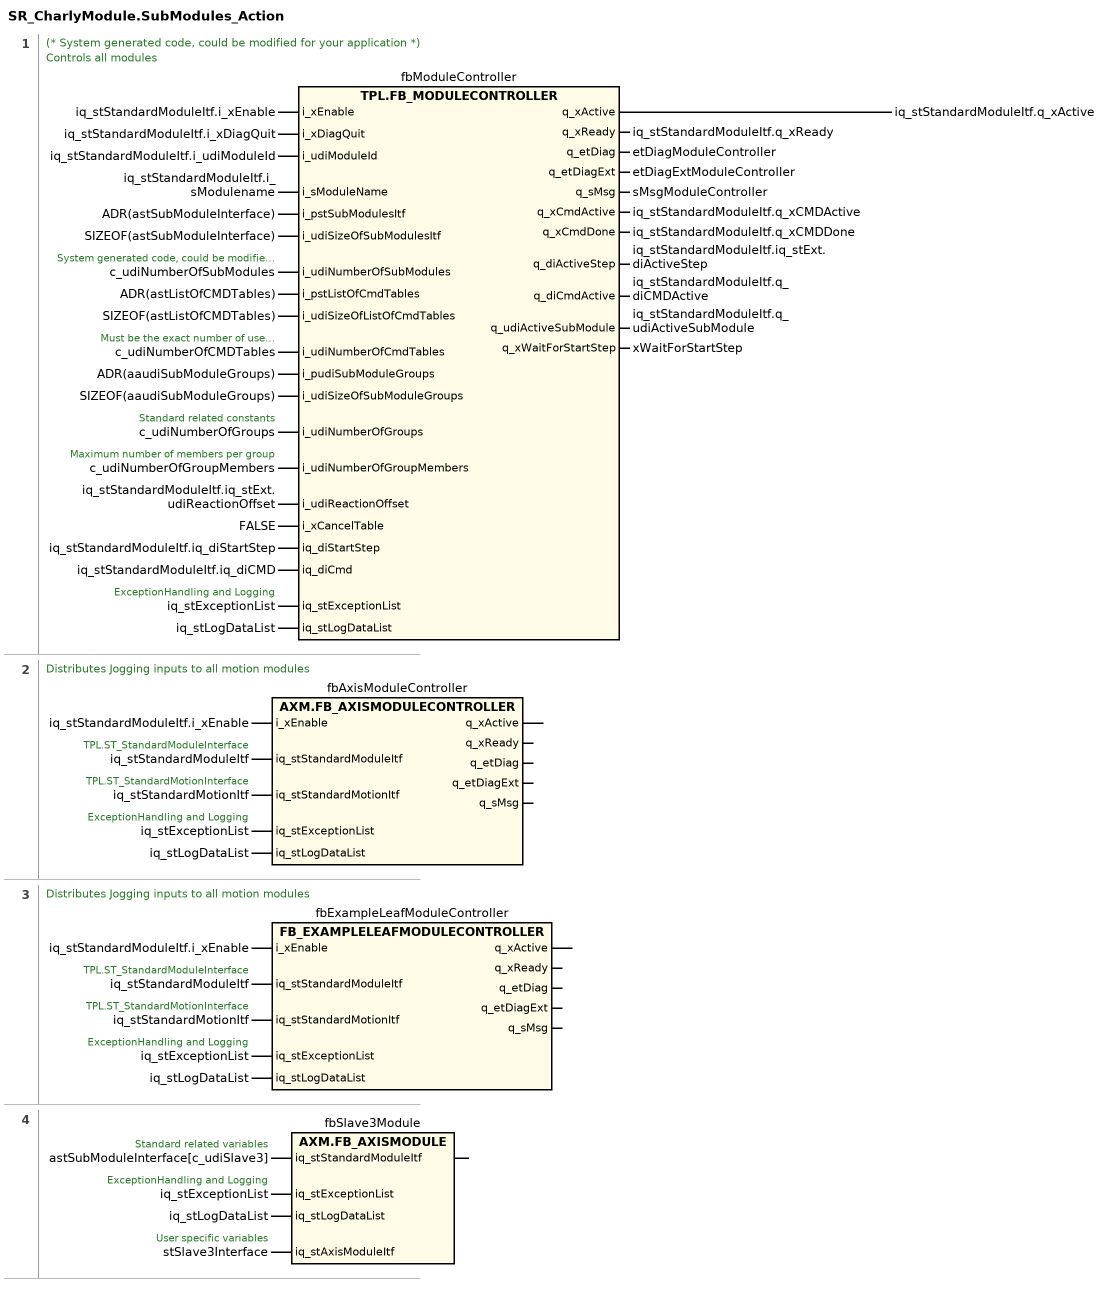
// NETWORK 1
// 					(* System generated code, could be modified for your application *)
// Controls all modules
//
//   fbModuleController: Modules related variables
//   c_udiNumberOfSubModules: System generated code, could be modified for your application
//   c_udiNumberOfCMDTables: Must be the exact number of used CMDTables!
//   c_udiNumberOfGroups: Standard related constants
//   c_udiNumberOfGroupMembers: Maximum number of members per group
//   iq_stExceptionList: ExceptionHandling and Logging
fbModuleController(
    i_xEnable := iq_stStandardModuleItf.i_xEnable,
    i_xDiagQuit := iq_stStandardModuleItf.i_xDiagQuit,
    i_udiModuleId := iq_stStandardModuleItf.i_udiModuleId,
    i_sModuleName := iq_stStandardModuleItf.i_sModulename,
    i_pstSubModulesItf := ADR(astSubModuleInterface),
    i_udiSizeOfSubModulesItf := SIZEOF(astSubModuleInterface),
    i_udiNumberOfSubModules := c_udiNumberOfSubModules,
    i_pstListOfCmdTables := ADR(astListOfCMDTables),
    i_udiSizeOfListOfCmdTables := SIZEOF(astListOfCMDTables),
    i_udiNumberOfCmdTables := c_udiNumberOfCMDTables,
    i_pudiSubModuleGroups := ADR(aaudiSubModuleGroups),
    i_udiSizeOfSubModuleGroups := SIZEOF(aaudiSubModuleGroups),
    i_udiNumberOfGroups := c_udiNumberOfGroups,
    i_udiNumberOfGroupMembers := c_udiNumberOfGroupMembers,
    i_udiReactionOffset := iq_stStandardModuleItf.iq_stExt.udiReactionOffset,
    i_xCancelTable := FALSE,
    iq_diStartStep := iq_stStandardModuleItf.iq_diStartStep,
    iq_diCmd := iq_stStandardModuleItf.iq_diCMD,
    iq_stExceptionList := iq_stExceptionList,
    iq_stLogDataList := iq_stLogDataList,
    q_xReady => iq_stStandardModuleItf.q_xReady,
    q_etDiag => etDiagModuleController,
    q_etDiagExt => etDiagExtModuleController,
    q_sMsg => sMsgModuleController,
    q_xCmdActive => iq_stStandardModuleItf.q_xCMDActive,
    q_xCmdDone => iq_stStandardModuleItf.q_xCMDDone,
    q_diActiveStep => iq_stStandardModuleItf.iq_stExt.diActiveStep,
    q_diCmdActive => iq_stStandardModuleItf.q_diCMDActive,
    q_udiActiveSubModule => iq_stStandardModuleItf.q_udiActiveSubModule,
    q_xWaitForStartStep => xWaitForStartStep); // TPL.FB_MODULECONTROLLER
iq_stStandardModuleItf.q_xActive := fbModuleController.q_xActive;

// NETWORK 2
// Distributes Jogging inputs to all motion modules
//   iq_stStandardModuleItf: TPL.ST_StandardModuleInterface
//   iq_stStandardMotionItf: TPL.ST_StandardMotionInterface
//   iq_stExceptionList: ExceptionHandling and Logging
fbAxisModuleController(
    i_xEnable := iq_stStandardModuleItf.i_xEnable,
    iq_stStandardModuleItf := iq_stStandardModuleItf,
    iq_stStandardMotionItf := iq_stStandardMotionItf,
    iq_stExceptionList := iq_stExceptionList,
    iq_stLogDataList := iq_stLogDataList); // AXM.FB_AXISMODULECONTROLLER

